gfCNCPoint6[3646] = {X 38.0615, Y 40.7422, Z -8.0000, A 0.000, B 0.000, C 0.000 }
gfCNCPoint6[3647] = {X 38.9310, Y 40.2409, Z -8.0000, A 0.000, B 0.000, C 0.000 }
gfCNCPoint6[3648] = {X 39.5220, Y 38.8450, Z -8.0000, A 0.000, B 0.000, C 0.000 }
gfCNCPoint6[3649] = {X 40.0631, Y 37.4290, Z -8.0000, A 0.000, B 0.000, C 0.000 }
gfCNCPoint6[3650] = {X 43.6474, Y 27.8074, Z -8.0000, A 0.000, B 0.000, C 0.000 }
gfCNCPoint6[3651] = {X 39.8991, Y 26.4111, Z -8.0000, A 0.000, B 0.000, C 0.000 }
gfCNCPoint6[3652] = {X 43.7224, Y 27.8353, Z -8.0000, A 0.000, B 0.000, C 0.000 }
gfCNCPoint6[3653] = {X 48.3793, Y 15.3344, Z -8.0000, A 0.000, B 0.000, C 0.000 }
gfCNCPoint6[3654] = {X 47.9922, Y 14.6130, Z -8.0000, A 0.000, B 0.000, C 0.000 }
gfCNCPoint6[3655] = {X 47.7508, Y 13.8307, Z -8.0000, A 0.000, B 0.000, C 0.000 }
gfCNCPoint6[3656] = {X 47.6644, Y 13.0166, Z -8.0000, A 0.000, B 0.000, C 0.000 }
gfCNCPoint6[3657] = {X 47.6642, Y 12.1868, Z -8.0000, A 0.000, B 0.000, C 0.000 }
gfCNCPoint6[3658] = {X 47.7705, Y 11.2433, Z -8.0000, A 0.000, B 0.000, C 0.000 }
gfCNCPoint6[3659] = {X 48.0841, Y 10.3472, Z -8.0000, A 0.000, B 0.000, C 0.000 }
gfCNCPoint6[3660] = {X 48.5893, Y 9.5432, Z -8.0000, A 0.000, B 0.000, C 0.000 }
gfCNCPoint6[3661] = {X 49.2606, Y 8.8719, Z -8.0000, A 0.000, B 0.000, C 0.000 }
gfCNCPoint6[3662] = {X 50.0646, Y 8.3667, Z -8.0000, A 0.000, B 0.000, C 0.000 }
gfCNCPoint6[3663] = {X 50.9607, Y 8.0531, Z -8.0000, A 0.000, B 0.000, C 0.000 }
gfCNCPoint6[3664] = {X 51.9042, Y 7.9468, Z -8.0000, A 0.000, B 0.000, C 0.000 }
gfCNCPoint6[3665] = {X 59.6221, Y 7.9468, Z -8.0000, A 0.000, B 0.000, C 0.000 }
gfCNCPoint6[3666] = {X 60.5656, Y 8.0531, Z -8.0000, A 0.000, B 0.000, C 0.000 }
gfCNCPoint6[3667] = {X 61.4618, Y 8.3667, Z -8.0000, A 0.000, B 0.000, C 0.000 }
gfCNCPoint6[3668] = {X 62.2657, Y 8.8718, Z -8.0000, A 0.000, B 0.000, C 0.000 }
gfCNCPoint6[3669] = {X 62.9371, Y 9.5432, Z -8.0000, A 0.000, B 0.000, C 0.000 }
gfCNCPoint6[3670] = {X 63.4422, Y 10.3471, Z -8.0000, A 0.000, B 0.000, C 0.000 }
gfCNCPoint6[3671] = {X 63.7558, Y 11.2433, Z -8.0000, A 0.000, B 0.000, C 0.000 }
gfCNCPoint6[3672] = {X 63.8621, Y 12.1868, Z -8.0000, A 0.000, B 0.000, C 0.000 }
gfCNCPoint6[3673] = {X 63.8621, Y 12.9782, Z -8.0000, A 0.000, B 0.000, C 0.000 }
gfCNCPoint6[3674] = {X 63.7772, Y 13.8222, Z -8.0000, A 0.000, B 0.000, C 0.000 }
gfCNCPoint6[3675] = {X 63.5261, Y 14.6323, Z -8.0000, A 0.000, B 0.000, C 0.000 }
gfCNCPoint6[3676] = {X 63.1187, Y 15.3763, Z -8.0000, A 0.000, B 0.000, C 0.000 }
gfCNCPoint6[3677] = {X 63.3523, Y 15.9915, Z -8.0000, A 0.000, B 0.000, C 0.000 }
gfCNCPoint6[3678] = {X 66.1652, Y 23.4578, Z -8.0000, A 0.000, B 0.000, C 0.000 }
gfCNCPoint6[3679] = {X 72.1363, Y 39.5291, Z -8.0000, A 0.000, B 0.000, C 0.000 }
gfCNCPoint6[3680] = {X 72.4543, Y 40.3288, Z -8.0000, A 0.000, B 0.000, C 0.000 }
gfCNCPoint6[3681] = {X 73.2915, Y 40.8190, Z -8.0000, A 0.000, B 0.000, C 0.000 }
gfCNCPoint6[3682] = {X 73.9953, Y 41.4867, Z -8.0000, A 0.000, B 0.000, C 0.000 }
gfCNCPoint6[3683] = {X 74.5289, Y 42.2969, Z -8.0000, A 0.000, B 0.000, C 0.000 }
gfCNCPoint6[3684] = {X 74.8645, Y 43.2072, Z -8.0000, A 0.000, B 0.000, C 0.000 }
gfCNCPoint6[3685] = {X 74.9843, Y 44.1699, Z -8.0000, A 0.000, B 0.000, C 0.000 }
gfCNCPoint6[3686] = {X 74.9845, Y 45.0000, Z -8.0000, A 0.000, B 0.000, C 0.000 }
gfCNCPoint6[3687] = {X 74.8782, Y 45.9435, Z -8.0000, A 0.000, B 0.000, C 0.000 }
gfCNCPoint6[3688] = {X 74.5646, Y 46.8397, Z -8.0000, A 0.000, B 0.000, C 0.000 }
gfCNCPoint6[3689] = {X 74.0594, Y 47.6436, Z -8.0000, A 0.000, B 0.000, C 0.000 }
gfCNCPoint6[3690] = {X 73.3881, Y 48.3150, Z -8.0000, A 0.000, B 0.000, C 0.000 }
gfCNCPoint6[3691] = {X 72.5841, Y 48.8201, Z -8.0000, A 0.000, B 0.000, C 0.000 }
gfCNCPoint6[3692] = {X 71.6879, Y 49.1337, Z -8.0000, A 0.000, B 0.000, C 0.000 }
gfCNCPoint6[3693] = {X 70.7445, Y 49.2400, Z -8.0000, A 0.000, B 0.000, C 0.000 }
gfCNCPoint6[3694] = {X 64.1851, Y 49.2400, Z -8.0000, A 0.000, B 0.000, C 0.000 }
gfCNCPoint6[3695] = {X 63.2416, Y 49.1337, Z -8.0000, A 0.000, B 0.000, C 0.000 }
gfCNCPoint6[3696] = {X 62.3455, Y 48.8201, Z -8.0000, A 0.000, B 0.000, C 0.000 }
gfCNCPoint6[3697] = {X 61.5415, Y 48.3150, Z -8.0000, A 0.000, B 0.000, C 0.000 }
gfCNCPoint6[3698] = {X 60.8702, Y 47.6436, Z -8.0000, A 0.000, B 0.000, C 0.000 }
gfCNCPoint6[3699] = {X 60.3650, Y 46.8397, Z -8.0000, A 0.000, B 0.000, C 0.000 }
gfCNCPoint6[3700] = {X 60.0514, Y 45.9435, Z -8.0000, A 0.000, B 0.000, C 0.000 }
gfCNCPoint6[3701] = {X 59.9451, Y 45.0000, Z -8.0000, A 0.000, B 0.000, C 0.000 }
gfCNCPoint6[3702] = {X 59.9451, Y 44.2085, Z -8.0000, A 0.000, B 0.000, C 0.000 }
gfCNCPoint6[3703] = {X 60.0327, Y 43.3528, Z -8.0000, A 0.000, B 0.000, C 0.000 }
gfCNCPoint6[3704] = {X 60.2911, Y 42.5324, Z -8.0000, A 0.000, B 0.000, C 0.000 }
gfCNCPoint6[3705] = {X 60.7098, Y 41.7810, Z -8.0000, A 0.000, B 0.000, C 0.000 }
gfCNCPoint6[3706] = {X 60.0623, Y 40.0092, Z -8.0000, A 0.000, B 0.000, C 0.000 }
gfCNCPoint6[3707] = {X 52.0229, Y 40.0092, Z -8.0000, A 0.000, B 0.000, C 0.000 }
gfCNCPoint6[3708] = {X 51.2471, Y 42.0939, Z -8.0000, A 0.000, B 0.000, C 0.000 }
gfCNCPoint6[3709] = {X 51.2689, Y 42.1309, Z -8.0000, A 0.000, B 0.000, C 0.000 }
gfCNCPoint6[3710] = {X 51.5641, Y 42.7777, Z -8.0000, A 0.000, B 0.000, C 0.000 }
gfCNCPoint6[3711] = {X 51.7471, Y 43.4647, Z -8.0000, A 0.000, B 0.000, C 0.000 }
gfCNCPoint6[3712] = {X 51.8128, Y 44.1726, Z -8.0000, A 0.000, B 0.000, C 0.000 }
gfCNCPoint6[3713] = {X 51.8129, Y 45.0000, Z -8.0000, A 0.000, B 0.000, C 0.000 }
gfCNCPoint6[3714] = {X 51.7066, Y 45.9435, Z -8.0000, A 0.000, B 0.000, C 0.000 }
gfCNCPoint6[3715] = {X 51.3930, Y 46.8397, Z -8.0000, A 0.000, B 0.000, C 0.000 }
gfCNCPoint6[3716] = {X 50.8879, Y 47.6436, Z -8.0000, A 0.000, B 0.000, C 0.000 }
gfCNCPoint6[3717] = {X 50.2165, Y 48.3150, Z -8.0000, A 0.000, B 0.000, C 0.000 }
gfCNCPoint6[3718] = {X 49.4126, Y 48.8201, Z -8.0000, A 0.000, B 0.000, C 0.000 }
gfCNCPoint6[3719] = {X 48.5164, Y 49.1337, Z -8.0000, A 0.000, B 0.000, C 0.000 }
gfCNCPoint6[3720] = {X 47.5729, Y 49.2400, Z -8.0000, A 0.000, B 0.000, C 0.000 }
gfCNCPoint6[3721] = {X 40.6393, Y 49.2400, Z -8.0000, A 0.000, B 0.000, C 0.000 }
gfCNCPoint6[3722] = {X 39.6958, Y 49.1337, Z -8.0000, A 0.000, B 0.000, C 0.000 }
gfCNCPoint6[3723] = {X 38.7996, Y 48.8201, Z -8.0000, A 0.000, B 0.000, C 0.000 }
gfCNCPoint6[3724] = {X 37.9957, Y 48.3150, Z -8.0000, A 0.000, B 0.000, C 0.000 }
gfCNCPoint6[3725] = {X 37.3243, Y 47.6436, Z -8.0000, A 0.000, B 0.000, C 0.000 }
gfCNCPoint6[3726] = {X 36.8192, Y 46.8397, Z -8.0000, A 0.000, B 0.000, C 0.000 }
gfCNCPoint6[3727] = {X 36.5056, Y 45.9435, Z -8.0000, A 0.000, B 0.000, C 0.000 }
gfCNCPoint6[3728] = {X 36.3993, Y 45.0000, Z -8.0000, A 0.000, B 0.000, C 0.000 }
gfCNCPoint6[3729] = {X 36.3993, Y 44.2086, Z -8.0000, A 0.000, B 0.000, C 0.000 }
gfCNCPoint6[3730] = {X 36.5152, Y 43.2242, Z -8.0000, A 0.000, B 0.000, C 0.000 }
gfCNCPoint6[3731] = {X 36.8565, Y 42.2936, Z -8.0000, A 0.000, B 0.000, C 0.000 }
gfCNCPoint6[3732] = {X 37.4045, Y 41.4677, Z -8.0000, A 0.000, B 0.000, C 0.000 }
gfCNCPoint6[3733] = {X 38.1293, Y 40.7916, Z -8.0000, A 0.000, B 0.000, C 0.000 }
gfCNCPoint6[3734] = {X 38.9913, Y 40.3022, Z -8.0000, A 0.000, B 0.000, C 0.000 }
gfCNCPoint6[3735] = {X 39.5904, Y 38.8895, Z -8.0000, A 0.000, B 0.000, C 0.000 }
gfCNCPoint6[3736] = {X 40.1384, Y 37.4563, Z -8.0000, A 0.000, B 0.000, C 0.000 }
gfCNCPoint6[3737] = {X 43.7224, Y 27.8353, Z -8.0000, A 0.000, B 0.000, C 0.000 }
gfCNCPoint6[3738] = {X 39.9740, Y 26.4390, Z -8.0000, A 0.000, B 0.000, C 0.000 }
gfCNCPoint6[3739] = {X 43.7974, Y 27.8633, Z -8.0000, A 0.000, B 0.000, C 0.000 }
gfCNCPoint6[3740] = {X 48.4687, Y 15.3238, Z -8.0000, A 0.000, B 0.000, C 0.000 }
gfCNCPoint6[3741] = {X 48.0765, Y 14.6072, Z -8.0000, A 0.000, B 0.000, C 0.000 }
gfCNCPoint6[3742] = {X 47.8320, Y 13.8279, Z -8.0000, A 0.000, B 0.000, C 0.000 }
gfCNCPoint6[3743] = {X 47.7444, Y 13.0158, Z -8.0000, A 0.000, B 0.000, C 0.000 }
gfCNCPoint6[3744] = {X 47.7442, Y 12.1868, Z -8.0000, A 0.000, B 0.000, C 0.000 }
gfCNCPoint6[3745] = {X 47.8485, Y 11.2611, Z -8.0000, A 0.000, B 0.000, C 0.000 }
gfCNCPoint6[3746] = {X 48.1562, Y 10.3819, Z -8.0000, A 0.000, B 0.000, C 0.000 }
gfCNCPoint6[3747] = {X 48.6518, Y 9.5931, Z -8.0000, A 0.000, B 0.000, C 0.000 }
gfCNCPoint6[3748] = {X 49.3105, Y 8.9344, Z -8.0000, A 0.000, B 0.000, C 0.000 }
gfCNCPoint6[3749] = {X 50.0993, Y 8.4388, Z -8.0000, A 0.000, B 0.000, C 0.000 }
gfCNCPoint6[3750] = {X 50.9785, Y 8.1311, Z -8.0000, A 0.000, B 0.000, C 0.000 }
gfCNCPoint6[3751] = {X 51.9042, Y 8.0268, Z -8.0000, A 0.000, B 0.000, C 0.000 }
gfCNCPoint6[3752] = {X 59.6221, Y 8.0268, Z -8.0000, A 0.000, B 0.000, C 0.000 }
gfCNCPoint6[3753] = {X 60.5478, Y 8.1311, Z -8.0000, A 0.000, B 0.000, C 0.000 }
gfCNCPoint6[3754] = {X 61.4271, Y 8.4388, Z -8.0000, A 0.000, B 0.000, C 0.000 }
gfCNCPoint6[3755] = {X 62.2158, Y 8.9344, Z -8.0000, A 0.000, B 0.000, C 0.000 }
gfCNCPoint6[3756] = {X 62.8745, Y 9.5931, Z -8.0000, A 0.000, B 0.000, C 0.000 }
gfCNCPoint6[3757] = {X 63.3702, Y 10.3819, Z -8.0000, A 0.000, B 0.000, C 0.000 }
gfCNCPoint6[3758] = {X 63.6778, Y 11.2611, Z -8.0000, A 0.000, B 0.000, C 0.000 }
gfCNCPoint6[3759] = {X 63.7821, Y 12.1868, Z -8.0000, A 0.000, B 0.000, C 0.000 }
gfCNCPoint6[3760] = {X 63.7821, Y 12.9782, Z -8.0000, A 0.000, B 0.000, C 0.000 }
gfCNCPoint6[3761] = {X 63.6961, Y 13.8198, Z -8.0000, A 0.000, B 0.000, C 0.000 }
gfCNCPoint6[3762] = {X 63.4415, Y 14.6267, Z -8.0000, A 0.000, B 0.000, C 0.000 }
gfCNCPoint6[3763] = {X 63.0289, Y 15.3654, Z -8.0000, A 0.000, B 0.000, C 0.000 }
gfCNCPoint6[3764] = {X 63.2774, Y 16.0198, Z -8.0000, A 0.000, B 0.000, C 0.000 }
gfCNCPoint6[3765] = {X 66.0903, Y 23.4859, Z -8.0000, A 0.000, B 0.000, C 0.000 }
gfCNCPoint6[3766] = {X 72.0617, Y 39.5578, Z -8.0000, A 0.000, B 0.000, C 0.000 }
gfCNCPoint6[3767] = {X 72.3921, Y 40.3890, Z -8.0000, A 0.000, B 0.000, C 0.000 }
gfCNCPoint6[3768] = {X 73.2225, Y 40.8674, Z -8.0000, A 0.000, B 0.000, C 0.000 }
gfCNCPoint6[3769] = {X 73.9214, Y 41.5231, Z -8.0000, A 0.000, B 0.000, C 0.000 }
gfCNCPoint6[3770] = {X 74.4516, Y 42.3213, Z -8.0000, A 0.000, B 0.000, C 0.000 }
gfCNCPoint6[3771] = {X 74.7852, Y 43.2197, Z -8.0000, A 0.000, B 0.000, C 0.000 }
gfCNCPoint6[3772] = {X 74.9043, Y 44.1706, Z -8.0000, A 0.000, B 0.000, C 0.000 }
gfCNCPoint6[3773] = {X 74.9045, Y 45.0000, Z -8.0000, A 0.000, B 0.000, C 0.000 }
gfCNCPoint6[3774] = {X 74.8002, Y 45.9257, Z -8.0000, A 0.000, B 0.000, C 0.000 }
gfCNCPoint6[3775] = {X 74.4925, Y 46.8050, Z -8.0000, A 0.000, B 0.000, C 0.000 }
gfCNCPoint6[3776] = {X 73.9969, Y 47.5937, Z -8.0000, A 0.000, B 0.000, C 0.000 }
gfCNCPoint6[3777] = {X 73.3382, Y 48.2524, Z -8.0000, A 0.000, B 0.000, C 0.000 }
gfCNCPoint6[3778] = {X 72.5494, Y 48.7480, Z -8.0000, A 0.000, B 0.000, C 0.000 }
gfCNCPoint6[3779] = {X 71.6701, Y 49.0557, Z -8.0000, A 0.000, B 0.000, C 0.000 }
gfCNCPoint6[3780] = {X 70.7445, Y 49.1600, Z -8.0000, A 0.000, B 0.000, C 0.000 }
gfCNCPoint6[3781] = {X 64.1851, Y 49.1600, Z -8.0000, A 0.000, B 0.000, C 0.000 }
gfCNCPoint6[3782] = {X 63.2594, Y 49.0557, Z -8.0000, A 0.000, B 0.000, C 0.000 }
gfCNCPoint6[3783] = {X 62.3802, Y 48.7480, Z -8.0000, A 0.000, B 0.000, C 0.000 }
gfCNCPoint6[3784] = {X 61.5914, Y 48.2524, Z -8.0000, A 0.000, B 0.000, C 0.000 }
gfCNCPoint6[3785] = {X 60.9327, Y 47.5937, Z -8.0000, A 0.000, B 0.000, C 0.000 }
gfCNCPoint6[3786] = {X 60.4371, Y 46.8050, Z -8.0000, A 0.000, B 0.000, C 0.000 }
gfCNCPoint6[3787] = {X 60.1294, Y 45.9257, Z -8.0000, A 0.000, B 0.000, C 0.000 }
gfCNCPoint6[3788] = {X 60.0251, Y 45.0000, Z -8.0000, A 0.000, B 0.000, C 0.000 }
gfCNCPoint6[3789] = {X 60.0251, Y 44.2086, Z -8.0000, A 0.000, B 0.000, C 0.000 }
gfCNCPoint6[3790] = {X 60.1139, Y 43.3555, Z -8.0000, A 0.000, B 0.000, C 0.000 }
gfCNCPoint6[3791] = {X 60.3756, Y 42.5387, Z -8.0000, A 0.000, B 0.000, C 0.000 }
gfCNCPoint6[3792] = {X 60.7994, Y 41.7930, Z -8.0000, A 0.000, B 0.000, C 0.000 }
gfCNCPoint6[3793] = {X 60.1182, Y 39.9292, Z -8.0000, A 0.000, B 0.000, C 0.000 }
gfCNCPoint6[3794] = {X 51.9673, Y 39.9292, Z -8.0000, A 0.000, B 0.000, C 0.000 }
gfCNCPoint6[3795] = {X 51.1588, Y 42.1017, Z -8.0000, A 0.000, B 0.000, C 0.000 }
gfCNCPoint6[3796] = {X 51.1995, Y 42.1708, Z -8.0000, A 0.000, B 0.000, C 0.000 }
gfCNCPoint6[3797] = {X 51.4890, Y 42.8052, Z -8.0000, A 0.000, B 0.000, C 0.000 }
gfCNCPoint6[3798] = {X 51.6684, Y 43.4790, Z -8.0000, A 0.000, B 0.000, C 0.000 }
gfCNCPoint6[3799] = {X 51.7328, Y 44.1733, Z -8.0000, A 0.000, B 0.000, C 0.000 }
gfCNCPoint6[3800] = {X 51.7329, Y 45.0000, Z -8.0000, A 0.000, B 0.000, C 0.000 }
gfCNCPoint6[3801] = {X 51.6286, Y 45.9257, Z -8.0000, A 0.000, B 0.000, C 0.000 }
gfCNCPoint6[3802] = {X 51.3210, Y 46.8050, Z -8.0000, A 0.000, B 0.000, C 0.000 }
gfCNCPoint6[3803] = {X 50.8253, Y 47.5937, Z -8.0000, A 0.000, B 0.000, C 0.000 }
gfCNCPoint6[3804] = {X 50.1666, Y 48.2524, Z -8.0000, A 0.000, B 0.000, C 0.000 }
gfCNCPoint6[3805] = {X 49.3779, Y 48.7480, Z -8.0000, A 0.000, B 0.000, C 0.000 }
gfCNCPoint6[3806] = {X 48.4986, Y 49.0557, Z -8.0000, A 0.000, B 0.000, C 0.000 }
gfCNCPoint6[3807] = {X 47.5729, Y 49.1600, Z -8.0000, A 0.000, B 0.000, C 0.000 }
gfCNCPoint6[3808] = {X 40.6393, Y 49.1600, Z -8.0000, A 0.000, B 0.000, C 0.000 }
gfCNCPoint6[3809] = {X 39.7136, Y 49.0557, Z -8.0000, A 0.000, B 0.000, C 0.000 }
gfCNCPoint6[3810] = {X 38.8343, Y 48.7480, Z -8.0000, A 0.000, B 0.000, C 0.000 }
gfCNCPoint6[3811] = {X 38.0456, Y 48.2524, Z -8.0000, A 0.000, B 0.000, C 0.000 }
gfCNCPoint6[3812] = {X 37.3869, Y 47.5937, Z -8.0000, A 0.000, B 0.000, C 0.000 }
gfCNCPoint6[3813] = {X 36.8913, Y 46.8050, Z -8.0000, A 0.000, B 0.000, C 0.000 }
gfCNCPoint6[3814] = {X 36.5836, Y 45.9257, Z -8.0000, A 0.000, B 0.000, C 0.000 }
gfCNCPoint6[3815] = {X 36.4793, Y 45.0000, Z -8.0000, A 0.000, B 0.000, C 0.000 }
gfCNCPoint6[3816] = {X 36.4793, Y 44.2086, Z -8.0000, A 0.000, B 0.000, C 0.000 }
gfCNCPoint6[3817] = {X 36.5945, Y 43.2366, Z -8.0000, A 0.000, B 0.000, C 0.000 }
gfCNCPoint6[3818] = {X 36.9336, Y 42.3185, Z -8.0000, A 0.000, B 0.000, C 0.000 }
gfCNCPoint6[3819] = {X 37.4778, Y 41.5050, Z -8.0000, A 0.000, B 0.000, C 0.000 }
gfCNCPoint6[3820] = {X 38.1970, Y 40.8412, Z -8.0000, A 0.000, B 0.000, C 0.000 }
gfCNCPoint6[3821] = {X 39.0514, Y 40.3638, Z -8.0000, A 0.000, B 0.000, C 0.000 }
gfCNCPoint6[3822] = {X 39.6586, Y 38.9342, Z -8.0000, A 0.000, B 0.000, C 0.000 }
gfCNCPoint6[3823] = {X 40.2136, Y 37.4835, Z -8.0000, A 0.000, B 0.000, C 0.000 }
gfCNCPoint6[3824] = {X 43.7974, Y 27.8633, Z -8.0000, A 0.000, B 0.000, C 0.000 }
gfCNCPoint6[3825] = {X 40.0490, Y 26.4669, Z -8.0000, A 0.000, B 0.000, C 0.000 }
gfCNCPoint6[3826] = {X 43.8723, Y 27.8912, Z -8.0000, A 0.000, B 0.000, C 0.000 }
gfCNCPoint6[3827] = {X 48.5582, Y 15.3126, Z -8.0000, A 0.000, B 0.000, C 0.000 }
gfCNCPoint6[3828] = {X 48.1610, Y 14.6012, Z -8.0000, A 0.000, B 0.000, C 0.000 }
gfCNCPoint6[3829] = {X 47.9131, Y 13.8250, Z -8.0000, A 0.000, B 0.000, C 0.000 }
gfCNCPoint6[3830] = {X 47.8244, Y 13.0151, Z -8.0000, A 0.000, B 0.000, C 0.000 }
gfCNCPoint6[3831] = {X 47.8242, Y 12.1868, Z -8.0000, A 0.000, B 0.000, C 0.000 }
gfCNCPoint6[3832] = {X 47.9265, Y 11.2789, Z -8.0000, A 0.000, B 0.000, C 0.000 }
gfCNCPoint6[3833] = {X 48.2283, Y 10.4166, Z -8.0000, A 0.000, B 0.000, C 0.000 }
gfCNCPoint6[3834] = {X 48.7144, Y 9.6430, Z -8.0000, A 0.000, B 0.000, C 0.000 }
gfCNCPoint6[3835] = {X 49.3604, Y 8.9969, Z -8.0000, A 0.000, B 0.000, C 0.000 }
gfCNCPoint6[3836] = {X 50.1340, Y 8.5109, Z -8.0000, A 0.000, B 0.000, C 0.000 }
gfCNCPoint6[3837] = {X 50.9963, Y 8.2091, Z -8.0000, A 0.000, B 0.000, C 0.000 }
gfCNCPoint6[3838] = {X 51.9042, Y 8.1068, Z -8.0000, A 0.000, B 0.000, C 0.000 }
gfCNCPoint6[3839] = {X 59.6221, Y 8.1068, Z -8.0000, A 0.000, B 0.000, C 0.000 }
gfCNCPoint6[3840] = {X 60.5300, Y 8.2091, Z -8.0000, A 0.000, B 0.000, C 0.000 }
gfCNCPoint6[3841] = {X 61.3924, Y 8.5109, Z -8.0000, A 0.000, B 0.000, C 0.000 }
gfCNCPoint6[3842] = {X 62.1660, Y 8.9969, Z -8.0000, A 0.000, B 0.000, C 0.000 }
gfCNCPoint6[3843] = {X 62.8120, Y 9.6430, Z -8.0000, A 0.000, B 0.000, C 0.000 }
gfCNCPoint6[3844] = {X 63.2981, Y 10.4166, Z -8.0000, A 0.000, B 0.000, C 0.000 }
gfCNCPoint6[3845] = {X 63.5998, Y 11.2789, Z -8.0000, A 0.000, B 0.000, C 0.000 }
gfCNCPoint6[3846] = {X 63.7021, Y 12.1868, Z -8.0000, A 0.000, B 0.000, C 0.000 }
gfCNCPoint6[3847] = {X 63.7021, Y 12.9782, Z -8.0000, A 0.000, B 0.000, C 0.000 }
gfCNCPoint6[3848] = {X 63.6148, Y 13.8174, Z -8.0000, A 0.000, B 0.000, C 0.000 }
gfCNCPoint6[3849] = {X 63.3568, Y 14.6208, Z -8.0000, A 0.000, B 0.000, C 0.000 }
gfCNCPoint6[3850] = {X 62.9390, Y 15.3539, Z -8.0000, A 0.000, B 0.000, C 0.000 }
gfCNCPoint6[3851] = {X 63.2026, Y 16.0481, Z -8.0000, A 0.000, B 0.000, C 0.000 }
gfCNCPoint6[3852] = {X 66.0153, Y 23.5139, Z -8.0000, A 0.000, B 0.000, C 0.000 }
gfCNCPoint6[3853] = {X 71.9870, Y 39.5865, Z -8.0000, A 0.000, B 0.000, C 0.000 }
gfCNCPoint6[3854] = {X 72.3301, Y 40.4495, Z -8.0000, A 0.000, B 0.000, C 0.000 }
gfCNCPoint6[3855] = {X 73.1536, Y 40.9160, Z -8.0000, A 0.000, B 0.000, C 0.000 }
gfCNCPoint6[3856] = {X 73.8474, Y 41.5597, Z -8.0000, A 0.000, B 0.000, C 0.000 }
gfCNCPoint6[3857] = {X 74.3743, Y 42.3459, Z -8.0000, A 0.000, B 0.000, C 0.000 }
gfCNCPoint6[3858] = {X 74.7059, Y 43.2324, Z -8.0000, A 0.000, B 0.000, C 0.000 }
gfCNCPoint6[3859] = {X 74.8243, Y 44.1714, Z -8.0000, A 0.000, B 0.000, C 0.000 }
gfCNCPoint6[3860] = {X 74.8245, Y 45.0000, Z -8.0000, A 0.000, B 0.000, C 0.000 }
gfCNCPoint6[3861] = {X 74.7222, Y 45.9079, Z -8.0000, A 0.000, B 0.000, C 0.000 }
gfCNCPoint6[3862] = {X 74.4204, Y 46.7702, Z -8.0000, A 0.000, B 0.000, C 0.000 }
gfCNCPoint6[3863] = {X 73.9343, Y 47.5438, Z -8.0000, A 0.000, B 0.000, C 0.000 }
gfCNCPoint6[3864] = {X 73.2883, Y 48.1899, Z -8.0000, A 0.000, B 0.000, C 0.000 }
gfCNCPoint6[3865] = {X 72.5147, Y 48.6760, Z -8.0000, A 0.000, B 0.000, C 0.000 }
gfCNCPoint6[3866] = {X 71.6523, Y 48.9777, Z -8.0000, A 0.000, B 0.000, C 0.000 }
gfCNCPoint6[3867] = {X 70.7445, Y 49.0800, Z -8.0000, A 0.000, B 0.000, C 0.000 }
gfCNCPoint6[3868] = {X 64.1851, Y 49.0800, Z -8.0000, A 0.000, B 0.000, C 0.000 }
gfCNCPoint6[3869] = {X 63.2772, Y 48.9777, Z -8.0000, A 0.000, B 0.000, C 0.000 }
gfCNCPoint6[3870] = {X 62.4149, Y 48.6760, Z -8.0000, A 0.000, B 0.000, C 0.000 }
gfCNCPoint6[3871] = {X 61.6413, Y 48.1899, Z -8.0000, A 0.000, B 0.000, C 0.000 }
gfCNCPoint6[3872] = {X 60.9953, Y 47.5438, Z -8.0000, A 0.000, B 0.000, C 0.000 }
gfCNCPoint6[3873] = {X 60.5092, Y 46.7702, Z -8.0000, A 0.000, B 0.000, C 0.000 }
gfCNCPoint6[3874] = {X 60.2074, Y 45.9079, Z -8.0000, A 0.000, B 0.000, C 0.000 }
gfCNCPoint6[3875] = {X 60.1051, Y 45.0000, Z -8.0000, A 0.000, B 0.000, C 0.000 }
gfCNCPoint6[3876] = {X 60.1051, Y 44.2086, Z -8.0000, A 0.000, B 0.000, C 0.000 }
gfCNCPoint6[3877] = {X 60.1950, Y 43.3582, Z -8.0000, A 0.000, B 0.000, C 0.000 }
gfCNCPoint6[3878] = {X 60.4602, Y 42.5452, Z -8.0000, A 0.000, B 0.000, C 0.000 }
gfCNCPoint6[3879] = {X 60.8891, Y 41.8054, Z -8.0000, A 0.000, B 0.000, C 0.000 }
gfCNCPoint6[3880] = {X 60.1742, Y 39.8492, Z -8.0000, A 0.000, B 0.000, C 0.000 }
gfCNCPoint6[3881] = {X 51.9117, Y 39.8492, Z -8.0000, A 0.000, B 0.000, C 0.000 }
gfCNCPoint6[3882] = {X 51.0705, Y 42.1095, Z -8.0000, A 0.000, B 0.000, C 0.000 }
gfCNCPoint6[3883] = {X 51.1302, Y 42.2107, Z -8.0000, A 0.000, B 0.000, C 0.000 }
gfCNCPoint6[3884] = {X 51.4139, Y 42.8327, Z -8.0000, A 0.000, B 0.000, C 0.000 }
gfCNCPoint6[3885] = {X 51.5897, Y 43.4933, Z -8.0000, A 0.000, B 0.000, C 0.000 }
gfCNCPoint6[3886] = {X 51.6528, Y 44.1740, Z -8.0000, A 0.000, B 0.000, C 0.000 }
gfCNCPoint6[3887] = {X 51.6529, Y 45.0000, Z -8.0000, A 0.000, B 0.000, C 0.000 }
gfCNCPoint6[3888] = {X 51.5506, Y 45.9079, Z -8.0000, A 0.000, B 0.000, C 0.000 }
gfCNCPoint6[3889] = {X 51.2489, Y 46.7702, Z -8.0000, A 0.000, B 0.000, C 0.000 }
gfCNCPoint6[3890] = {X 50.7628, Y 47.5438, Z -8.0000, A 0.000, B 0.000, C 0.000 }
gfCNCPoint6[3891] = {X 50.1168, Y 48.1899, Z -8.0000, A 0.000, B 0.000, C 0.000 }
gfCNCPoint6[3892] = {X 49.3432, Y 48.6760, Z -8.0000, A 0.000, B 0.000, C 0.000 }
gfCNCPoint6[3893] = {X 48.4808, Y 48.9777, Z -8.0000, A 0.000, B 0.000, C 0.000 }
gfCNCPoint6[3894] = {X 47.5729, Y 49.0800, Z -8.0000, A 0.000, B 0.000, C 0.000 }
gfCNCPoint6[3895] = {X 40.6393, Y 49.0800, Z -8.0000, A 0.000, B 0.000, C 0.000 }
gfCNCPoint6[3896] = {X 39.7314, Y 48.9777, Z -8.0000, A 0.000, B 0.000, C 0.000 }
gfCNCPoint6[3897] = {X 38.8691, Y 48.6760, Z -8.0000, A 0.000, B 0.000, C 0.000 }
gfCNCPoint6[3898] = {X 38.0955, Y 48.1899, Z -8.0000, A 0.000, B 0.000, C 0.000 }
gfCNCPoint6[3899] = {X 37.4494, Y 47.5438, Z -8.0000, A 0.000, B 0.000, C 0.000 }
gfCNCPoint6[3900] = {X 36.9633, Y 46.7702, Z -8.0000, A 0.000, B 0.000, C 0.000 }
gfCNCPoint6[3901] = {X 36.6616, Y 45.9079, Z -8.0000, A 0.000, B 0.000, C 0.000 }
gfCNCPoint6[3902] = {X 36.5593, Y 45.0000, Z -8.0000, A 0.000, B 0.000, C 0.000 }
gfCNCPoint6[3903] = {X 36.5593, Y 44.2086, Z -8.0000, A 0.000, B 0.000, C 0.000 }
gfCNCPoint6[3904] = {X 36.6733, Y 43.2512, Z -8.0000, A 0.000, B 0.000, C 0.000 }
gfCNCPoint6[3905] = {X 37.0087, Y 42.3474, Z -8.0000, A 0.000, B 0.000, C 0.000 }
gfCNCPoint6[3906] = {X 37.5468, Y 41.5474, Z -8.0000, A 0.000, B 0.000, C 0.000 }
gfCNCPoint6[3907] = {X 38.2576, Y 40.8961, Z -8.0000, A 0.000, B 0.000, C 0.000 }
gfCNCPoint6[3908] = {X 39.1014, Y 40.4297, Z -8.0000, A 0.000, B 0.000, C 0.000 }
gfCNCPoint6[3909] = {X 39.1158, Y 40.4158, Z -8.0000, A 0.000, B 0.000, C 0.000 }
gfCNCPoint6[3910] = {X 39.1244, Y 40.3964, Z -8.0000, A 0.000, B 0.000, C 0.000 }
gfCNCPoint6[3911] = {X 39.7328, Y 38.9641, Z -8.0000, A 0.000, B 0.000, C 0.000 }
gfCNCPoint6[3912] = {X 40.2888, Y 37.5107, Z -8.0000, A 0.000, B 0.000, C 0.000 }
gfCNCPoint6[3913] = {X 43.8723, Y 27.8912, Z -8.0000, A 0.000, B 0.000, C 0.000 }
gfCNCPoint6[3914] = {X 40.1240, Y 26.4948, Z -8.0000, A 0.000, B 0.000, C 0.000 }
gfCNCPoint6[3915] = {X 43.9473, Y 27.9191, Z -8.0000, A 0.000, B 0.000, C 0.000 }
gfCNCPoint6[3916] = {X 48.6479, Y 15.3010, Z -8.0000, A 0.000, B 0.000, C 0.000 }
gfCNCPoint6[3917] = {X 48.2407, Y 14.5838, Z -8.0000, A 0.000, B 0.000, C 0.000 }
gfCNCPoint6[3918] = {X 47.9892, Y 13.7983, Z -8.0000, A 0.000, B 0.000, C 0.000 }
gfCNCPoint6[3919] = {X 47.9042, Y 12.9780, Z -8.0000, A 0.000, B 0.000, C 0.000 }
gfCNCPoint6[3920] = {X 47.9042, Y 12.1868, Z -8.0000, A 0.000, B 0.000, C 0.000 }
gfCNCPoint6[3921] = {X 48.0045, Y 11.2967, Z -8.0000, A 0.000, B 0.000, C 0.000 }
gfCNCPoint6[3922] = {X 48.3003, Y 10.4513, Z -8.0000, A 0.000, B 0.000, C 0.000 }
gfCNCPoint6[3923] = {X 48.7769, Y 9.6929, Z -8.0000, A 0.000, B 0.000, C 0.000 }
gfCNCPoint6[3924] = {X 49.4103, Y 9.0595, Z -8.0000, A 0.000, B 0.000, C 0.000 }
gfCNCPoint6[3925] = {X 50.1687, Y 8.5829, Z -8.0000, A 0.000, B 0.000, C 0.000 }
gfCNCPoint6[3926] = {X 51.0141, Y 8.2871, Z -8.0000, A 0.000, B 0.000, C 0.000 }
gfCNCPoint6[3927] = {X 51.9042, Y 8.1868, Z -8.0000, A 0.000, B 0.000, C 0.000 }
gfCNCPoint6[3928] = {X 59.6221, Y 8.1868, Z -8.0000, A 0.000, B 0.000, C 0.000 }
gfCNCPoint6[3929] = {X 60.5122, Y 8.2871, Z -8.0000, A 0.000, B 0.000, C 0.000 }
gfCNCPoint6[3930] = {X 61.3577, Y 8.5829, Z -8.0000, A 0.000, B 0.000, C 0.000 }
gfCNCPoint6[3931] = {X 62.1161, Y 9.0595, Z -8.0000, A 0.000, B 0.000, C 0.000 }
gfCNCPoint6[3932] = {X 62.7495, Y 9.6929, Z -8.0000, A 0.000, B 0.000, C 0.000 }
gfCNCPoint6[3933] = {X 63.2260, Y 10.4513, Z -8.0000, A 0.000, B 0.000, C 0.000 }
gfCNCPoint6[3934] = {X 63.5218, Y 11.2967, Z -8.0000, A 0.000, B 0.000, C 0.000 }
gfCNCPoint6[3935] = {X 63.6221, Y 12.1868, Z -8.0000, A 0.000, B 0.000, C 0.000 }
gfCNCPoint6[3936] = {X 63.6219, Y 13.0192, Z -8.0000, A 0.000, B 0.000, C 0.000 }
gfCNCPoint6[3937] = {X 63.5278, Y 13.8416, Z -8.0000, A 0.000, B 0.000, C 0.000 }
gfCNCPoint6[3938] = {X 63.2664, Y 14.6271, Z -8.0000, A 0.000, B 0.000, C 0.000 }
gfCNCPoint6[3939] = {X 62.8489, Y 15.3419, Z -8.0000, A 0.000, B 0.000, C 0.000 }
gfCNCPoint6[3940] = {X 63.1278, Y 16.0764, Z -8.0000, A 0.000, B 0.000, C 0.000 }
gfCNCPoint6[3941] = {X 65.9404, Y 23.5419, Z -8.0000, A 0.000, B 0.000, C 0.000 }
gfCNCPoint6[3942] = {X 71.9123, Y 39.6152, Z -8.0000, A 0.000, B 0.000, C 0.000 }
gfCNCPoint6[3943] = {X 72.2607, Y 40.4916, Z -8.0000, A 0.000, B 0.000, C 0.000 }
gfCNCPoint6[3944] = {X 72.2711, Y 40.5075, Z -8.0000, A 0.000, B 0.000, C 0.000 }
gfCNCPoint6[3945] = {X 72.2868, Y 40.5181, Z -8.0000, A 0.000, B 0.000, C 0.000 }
gfCNCPoint6[3946] = {X 72.3497, Y 40.5450, Z -8.0000, A 0.000, B 0.000, C 0.000 }
gfCNCPoint6[3947] = {X 72.4122, Y 40.5731, Z -8.0000, A 0.000, B 0.000, C 0.000 }
gfCNCPoint6[3948] = {X 73.1913, Y 41.0445, Z -8.0000, A 0.000, B 0.000, C 0.000 }
gfCNCPoint6[3949] = {X 73.8436, Y 41.6799, Z -8.0000, A 0.000, B 0.000, C 0.000 }
gfCNCPoint6[3950] = {X 74.3353, Y 42.4464, Z -8.0000, A 0.000, B 0.000, C 0.000 }
gfCNCPoint6[3951] = {X 74.6408, Y 43.3042, Z -8.0000, A 0.000, B 0.000, C 0.000 }
gfCNCPoint6[3952] = {X 74.7445, Y 44.2089, Z -8.0000, A 0.000, B 0.000, C 0.000 }
gfCNCPoint6[3953] = {X 74.7445, Y 45.0000, Z -8.0000, A 0.000, B 0.000, C 0.000 }
gfCNCPoint6[3954] = {X 74.6442, Y 45.8901, Z -8.0000, A 0.000, B 0.000, C 0.000 }
gfCNCPoint6[3955] = {X 74.3483, Y 46.7355, Z -8.0000, A 0.000, B 0.000, C 0.000 }
gfCNCPoint6[3956] = {X 73.8718, Y 47.4940, Z -8.0000, A 0.000, B 0.000, C 0.000 }
gfCNCPoint6[3957] = {X 73.2384, Y 48.1273, Z -8.0000, A 0.000, B 0.000, C 0.000 }
gfCNCPoint6[3958] = {X 72.4800, Y 48.6039, Z -8.0000, A 0.000, B 0.000, C 0.000 }
gfCNCPoint6[3959] = {X 71.6345, Y 48.8997, Z -8.0000, A 0.000, B 0.000, C 0.000 }
gfCNCPoint6[3960] = {X 70.7445, Y 49.0000, Z -8.0000, A 0.000, B 0.000, C 0.000 }
gfCNCPoint6[3961] = {X 64.1851, Y 49.0000, Z -8.0000, A 0.000, B 0.000, C 0.000 }
gfCNCPoint6[3962] = {X 63.2951, Y 48.8997, Z -8.0000, A 0.000, B 0.000, C 0.000 }
gfCNCPoint6[3963] = {X 62.4496, Y 48.6039, Z -8.0000, A 0.000, B 0.000, C 0.000 }
gfCNCPoint6[3964] = {X 61.6912, Y 48.1273, Z -8.0000, A 0.000, B 0.000, C 0.000 }
gfCNCPoint6[3965] = {X 61.0578, Y 47.4940, Z -8.0000, A 0.000, B 0.000, C 0.000 }
gfCNCPoint6[3966] = {X 60.5813, Y 46.7355, Z -8.0000, A 0.000, B 0.000, C 0.000 }
gfCNCPoint6[3967] = {X 60.2854, Y 45.8901, Z -8.0000, A 0.000, B 0.000, C 0.000 }
gfCNCPoint6[3968] = {X 60.1851, Y 45.0000, Z -8.0000, A 0.000, B 0.000, C 0.000 }
gfCNCPoint6[3969] = {X 60.1855, Y 44.1538, Z -8.0000, A 0.000, B 0.000, C 0.000 }
gfCNCPoint6[3970] = {X 60.2746, Y 43.3674, Z -8.0000, A 0.000, B 0.000, C 0.000 }
gfCNCPoint6[3971] = {X 60.5168, Y 42.6140, Z -8.0000, A 0.000, B 0.000, C 0.000 }
gfCNCPoint6[3972] = {X 60.9025, Y 41.9231, Z -8.0000, A 0.000, B 0.000, C 0.000 }
gfCNCPoint6[3973] = {X 60.9788, Y 41.8179, Z -8.0000, A 0.000, B 0.000, C 0.000 }
gfCNCPoint6[3974] = {X 60.2301, Y 39.7692, Z -8.0000, A 0.000, B 0.000, C 0.000 }
gfCNCPoint6[3975] = {X 51.8432, Y 39.7692, Z -8.0000, A 0.000, B 0.000, C 0.000 }
gfCNCPoint6[3976] = {X 51.8432, Y 39.8040, Z -8.0000, A 0.000, B 0.000, C 0.000 }
gfCNCPoint6[3977] = {X 50.9823, Y 42.1173, Z -8.0000, A 0.000, B 0.000, C 0.000 }
gfCNCPoint6[3978] = {X 51.0732, Y 42.2728, Z -8.0000, A 0.000, B 0.000, C 0.000 }
gfCNCPoint6[3979] = {X 51.3482, Y 42.8869, Z -8.0000, A 0.000, B 0.000, C 0.000 }
gfCNCPoint6[3980] = {X 51.5164, Y 43.5384, Z -8.0000, A 0.000, B 0.000, C 0.000 }
gfCNCPoint6[3981] = {X 51.5729, Y 44.2089, Z -8.0000, A 0.000, B 0.000, C 0.000 }
gfCNCPoint6[3982] = {X 51.5729, Y 45.0000, Z -8.0000, A 0.000, B 0.000, C 0.000 }
gfCNCPoint6[3983] = {X 51.4726, Y 45.8901, Z -8.0000, A 0.000, B 0.000, C 0.000 }
gfCNCPoint6[3984] = {X 51.1768, Y 46.7355, Z -8.0000, A 0.000, B 0.000, C 0.000 }
gfCNCPoint6[3985] = {X 50.7003, Y 47.4940, Z -8.0000, A 0.000, B 0.000, C 0.000 }
gfCNCPoint6[3986] = {X 50.0669, Y 48.1273, Z -8.0000, A 0.000, B 0.000, C 0.000 }
gfCNCPoint6[3987] = {X 49.3085, Y 48.6039, Z -8.0000, A 0.000, B 0.000, C 0.000 }
gfCNCPoint6[3988] = {X 48.4630, Y 48.8997, Z -8.0000, A 0.000, B 0.000, C 0.000 }
gfCNCPoint6[3989] = {X 47.5729, Y 49.0000, Z -8.0000, A 0.000, B 0.000, C 0.000 }
gfCNCPoint6[3990] = {X 40.6393, Y 49.0000, Z -8.0000, A 0.000, B 0.000, C 0.000 }
gfCNCPoint6[3991] = {X 39.7492, Y 48.8997, Z -8.0000, A 0.000, B 0.000, C 0.000 }
gfCNCPoint6[3992] = {X 38.9038, Y 48.6039, Z -8.0000, A 0.000, B 0.000, C 0.000 }
gfCNCPoint6[3993] = {X 38.1453, Y 48.1273, Z -8.0000, A 0.000, B 0.000, C 0.000 }
gfCNCPoint6[3994] = {X 37.5120, Y 47.4940, Z -8.0000, A 0.000, B 0.000, C 0.000 }
gfCNCPoint6[3995] = {X 37.0354, Y 46.7355, Z -8.0000, A 0.000, B 0.000, C 0.000 }
gfCNCPoint6[3996] = {X 36.7396, Y 45.8901, Z -8.0000, A 0.000, B 0.000, C 0.000 }
gfCNCPoint6[3997] = {X 36.6393, Y 45.0000, Z -8.0000, A 0.000, B 0.000, C 0.000 }
gfCNCPoint6[3998] = {X 36.6397, Y 44.1538, Z -8.0000, A 0.000, B 0.000, C 0.000 }
gfCNCPoint6[3999] = {X 36.7563, Y 43.2486, Z -8.0000, A 0.000, B 0.000, C 0.000 }
gfCNCPoint6[4000] = {X 37.0750, Y 42.3933, Z -8.0000, A 0.000, B 0.000, C 0.000 }
gfCNCPoint6[4001] = {X 37.5793, Y 41.6327, Z -8.0000, A 0.000, B 0.000, C 0.000 }
gfCNCPoint6[4002] = {X 38.2429, Y 41.0061, Z -8.0000, A 0.000, B 0.000, C 0.000 }
gfCNCPoint6[4003] = {X 39.0313, Y 40.5462, Z -8.0000, A 0.000, B 0.000, C 0.000 }
gfCNCPoint6[4004] = {X 39.0813, Y 40.5247, Z -8.0000, A 0.000, B 0.000, C 0.000 }
gfCNCPoint6[4005] = {X 39.1315, Y 40.5038, Z -8.0000, A 0.000, B 0.000, C 0.000 }
gfCNCPoint6[4006] = {X 39.1655, Y 40.4817, Z -8.0000, A 0.000, B 0.000, C 0.000 }
gfCNCPoint6[4007] = {X 39.1888, Y 40.4485, Z -8.0000, A 0.000, B 0.000, C 0.000 }
gfCNCPoint6[4008] = {X 39.2125, Y 40.3954, Z -8.0000, A 0.000, B 0.000, C 0.000 }
gfCNCPoint6[4009] = {X 39.2361, Y 40.3422, Z -8.0000, A 0.000, B 0.000, C 0.000 }
gfCNCPoint6[4010] = {X 39.8247, Y 38.9502, Z -8.0000, A 0.000, B 0.000, C 0.000 }
gfCNCPoint6[4011] = {X 40.3639, Y 37.5383, Z -8.0000, A 0.000, B 0.000, C 0.000 }
gfCNCPoint6[4012] = {X 43.9473, Y 27.9191, Z -8.0000, A 0.000, B 0.000, C 0.000 }
gfCNCPoint6[4013] = {X 40.1240, Y 26.4948, Z -8.0000, A 0.000, B 0.000, C 0.000 }
gfCNCPoint6[4014] = {X 40.1240, Y 26.4948, Z -5.0000, A 0.000, B 0.000, C 0.000 }
gfCNCPoint6[4015] = {X 40.1240, Y 26.4948, Z 11.0000, A 0.000, B 0.000, C 0.000 }
gfCNCPoint6[4016] = {X 79.0216, Y 28.5909, Z 11.0000, A 0.000, B 0.000, C 0.000 }
gfCNCPoint6[4017] = {X 79.0216, Y 28.5909, Z -5.0000, A 0.000, B 0.000, C 0.000 }
gfCNCPoint6[4018] = {X 79.0216, Y 28.5909, Z -8.0000, A 0.000, B 0.000, C 0.000 }
gfCNCPoint6[4019] = {X 83.1016, Y 28.5909, Z -8.0000, A 0.000, B 0.000, C 0.000 }
gfCNCPoint6[4020] = {X 83.1017, Y 16.2734, Z -8.0000, A 0.000, B 0.000, C 0.000 }
gfCNCPoint6[4021] = {X 82.4635, Y 15.6023, Z -8.0000, A 0.000, B 0.000, C 0.000 }
gfCNCPoint6[4022] = {X 81.9830, Y 14.8106, Z -8.0000, A 0.000, B 0.000, C 0.000 }
gfCNCPoint6[4023] = {X 81.6823, Y 13.9347, Z -8.0000, A 0.000, B 0.000, C 0.000 }
gfCNCPoint6[4024] = {X 81.5752, Y 13.0148, Z -8.0000, A 0.000, B 0.000, C 0.000 }
gfCNCPoint6[4025] = {X 81.5751, Y 12.1868, Z -8.0000, A 0.000, B 0.000, C 0.000 }
gfCNCPoint6[4026] = {X 81.6834, Y 11.2255, Z -8.0000, A 0.000, B 0.000, C 0.000 }
gfCNCPoint6[4027] = {X 82.0029, Y 10.3124, Z -8.0000, A 0.000, B 0.000, C 0.000 }
gfCNCPoint6[4028] = {X 82.5176, Y 9.4933, Z -8.0000, A 0.000, B 0.000, C 0.000 }
gfCNCPoint6[4029] = {X 83.2016, Y 8.8093, Z -8.0000, A 0.000, B 0.000, C 0.000 }
gfCNCPoint6[4030] = {X 84.0207, Y 8.2946, Z -8.0000, A 0.000, B 0.000, C 0.000 }
gfCNCPoint6[4031] = {X 84.9338, Y 7.9751, Z -8.0000, A 0.000, B 0.000, C 0.000 }
gfCNCPoint6[4032] = {X 85.8951, Y 7.8668, Z -8.0000, A 0.000, B 0.000, C 0.000 }
gfCNCPoint6[4033] = {X 94.0497, Y 7.8668, Z -8.0000, A 0.000, B 0.000, C 0.000 }
gfCNCPoint6[4034] = {X 95.0110, Y 7.9751, Z -8.0000, A 0.000, B 0.000, C 0.000 }
gfCNCPoint6[4035] = {X 95.9240, Y 8.2946, Z -8.0000, A 0.000, B 0.000, C 0.000 }
gfCNCPoint6[4036] = {X 96.7431, Y 8.8093, Z -8.0000, A 0.000, B 0.000, C 0.000 }
gfCNCPoint6[4037] = {X 97.4272, Y 9.4933, Z -8.0000, A 0.000, B 0.000, C 0.000 }
gfCNCPoint6[4038] = {X 97.9419, Y 10.3124, Z -8.0000, A 0.000, B 0.000, C 0.000 }
gfCNCPoint6[4039] = {X 98.2614, Y 11.2255, Z -8.0000, A 0.000, B 0.000, C 0.000 }
gfCNCPoint6[4040] = {X 98.3697, Y 12.1868, Z -8.0000, A 0.000, B 0.000, C 0.000 }
gfCNCPoint6[4041] = {X 98.3697, Y 12.9782, Z -8.0000, A 0.000, B 0.000, C 0.000 }
gfCNCPoint6[4042] = {X 98.2968, Y 13.7675, Z -8.0000, A 0.000, B 0.000, C 0.000 }
gfCNCPoint6[4043] = {X 98.0809, Y 14.5303, Z -8.0000, A 0.000, B 0.000, C 0.000 }
gfCNCPoint6[4044] = {X 97.7293, Y 15.2407, Z -8.0000, A 0.000, B 0.000, C 0.000 }
gfCNCPoint6[4045] = {X 101.8771, Y 25.5237, Z -8.0000, A 0.000, B 0.000, C 0.000 }
gfCNCPoint6[4046] = {X 106.0160, Y 15.2206, Z -8.0000, A 0.000, B 0.000, C 0.000 }
gfCNCPoint6[4047] = {X 105.6759, Y 14.5280, Z -8.0000, A 0.000, B 0.000, C 0.000 }
gfCNCPoint6[4048] = {X 105.4645, Y 13.7858, Z -8.0000, A 0.000, B 0.000, C 0.000 }
gfCNCPoint6[4049] = {X 105.3885, Y 13.0179, Z -8.0000, A 0.000, B 0.000, C 0.000 }
gfCNCPoint6[4050] = {X 105.3883, Y 12.1868, Z -8.0000, A 0.000, B 0.000, C 0.000 }
gfCNCPoint6[4051] = {X 105.4966, Y 11.2255, Z -8.0000, A 0.000, B 0.000, C 0.000 }
gfCNCPoint6[4052] = {X 105.8161, Y 10.3124, Z -8.0000, A 0.000, B 0.000, C 0.000 }
gfCNCPoint6[4053] = {X 106.3308, Y 9.4933, Z -8.0000, A 0.000, B 0.000, C 0.000 }
gfCNCPoint6[4054] = {X 107.0148, Y 8.8093, Z -8.0000, A 0.000, B 0.000, C 0.000 }
gfCNCPoint6[4055] = {X 107.8339, Y 8.2946, Z -8.0000, A 0.000, B 0.000, C 0.000 }
gfCNCPoint6[4056] = {X 108.7470, Y 7.9751, Z -8.0000, A 0.000, B 0.000, C 0.000 }
gfCNCPoint6[4057] = {X 109.7083, Y 7.8668, Z -8.0000, A 0.000, B 0.000, C 0.000 }
gfCNCPoint6[4058] = {X 117.7916, Y 7.8668, Z -8.0000, A 0.000, B 0.000, C 0.000 }
gfCNCPoint6[4059] = {X 118.7529, Y 7.9751, Z -8.0000, A 0.000, B 0.000, C 0.000 }
gfCNCPoint6[4060] = {X 119.6660, Y 8.2946, Z -8.0000, A 0.000, B 0.000, C 0.000 }
gfCNCPoint6[4061] = {X 120.4851, Y 8.8093, Z -8.0000, A 0.000, B 0.000, C 0.000 }
gfCNCPoint6[4062] = {X 121.1691, Y 9.4933, Z -8.0000, A 0.000, B 0.000, C 0.000 }
gfCNCPoint6[4063] = {X 121.6838, Y 10.3124, Z -8.0000, A 0.000, B 0.000, C 0.000 }
gfCNCPoint6[4064] = {X 122.0033, Y 11.2255, Z -8.0000, A 0.000, B 0.000, C 0.000 }
gfCNCPoint6[4065] = {X 122.1116, Y 12.1868, Z -8.0000, A 0.000, B 0.000, C 0.000 }
gfCNCPoint6[4066] = {X 122.1116, Y 12.9782, Z -8.0000, A 0.000, B 0.000, C 0.000 }
gfCNCPoint6[4067] = {X 122.0103, Y 13.9078, Z -8.0000, A 0.000, B 0.000, C 0.000 }
gfCNCPoint6[4068] = {X 121.7114, Y 14.7939, Z -8.0000, A 0.000, B 0.000, C 0.000 }
gfCNCPoint6[4069] = {X 121.2288, Y 15.5949, Z -8.0000, A 0.000, B 0.000, C 0.000 }
gfCNCPoint6[4070] = {X 120.5851, Y 16.2732, Z -8.0000, A 0.000, B 0.000, C 0.000 }
gfCNCPoint6[4071] = {X 120.5853, Y 40.9148, Z -8.0000, A 0.000, B 0.000, C 0.000 }
gfCNCPoint6[4072] = {X 120.6230, Y 40.9460, Z -8.0000, A 0.000, B 0.000, C 0.000 }
gfCNCPoint6[4073] = {X 121.2460, Y 41.6147, Z -8.0000, A 0.000, B 0.000, C 0.000 }
gfCNCPoint6[4074] = {X 121.7145, Y 42.3996, Z -8.0000, A 0.000, B 0.000, C 0.000 }
gfCNCPoint6[4075] = {X 122.0073, Y 43.2654, Z -8.0000, A 0.000, B 0.000, C 0.000 }
gfCNCPoint6[4076] = {X 122.1114, Y 44.1734, Z -8.0000, A 0.000, B 0.000, C 0.000 }
gfCNCPoint6[4077] = {X 122.1116, Y 45.0000, Z -8.0000, A 0.000, B 0.000, C 0.000 }
gfCNCPoint6[4078] = {X 122.0033, Y 45.9613, Z -8.0000, A 0.000, B 0.000, C 0.000 }
gfCNCPoint6[4079] = {X 121.6838, Y 46.8744, Z -8.0000, A 0.000, B 0.000, C 0.000 }
gfCNCPoint6[4080] = {X 121.1691, Y 47.6935, Z -8.0000, A 0.000, B 0.000, C 0.000 }
gfCNCPoint6[4081] = {X 120.4851, Y 48.3775, Z -8.0000, A 0.000, B 0.000, C 0.000 }
gfCNCPoint6[4082] = {X 119.6660, Y 48.8922, Z -8.0000, A 0.000, B 0.000, C 0.000 }
gfCNCPoint6[4083] = {X 118.7529, Y 49.2117, Z -8.0000, A 0.000, B 0.000, C 0.000 }
gfCNCPoint6[4084] = {X 117.7916, Y 49.3200, Z -8.0000, A 0.000, B 0.000, C 0.000 }
gfCNCPoint6[4085] = {X 111.9185, Y 49.3200, Z -8.0000, A 0.000, B 0.000, C 0.000 }
gfCNCPoint6[4086] = {X 110.9619, Y 49.2128, Z -8.0000, A 0.000, B 0.000, C 0.000 }
gfCNCPoint6[4087] = {X 110.0529, Y 48.8964, Z -8.0000, A 0.000, B 0.000, C 0.000 }
gfCNCPoint6[4088] = {X 109.2365, Y 48.3866, Z -8.0000, A 0.000, B 0.000, C 0.000 }
gfCNCPoint6[4089] = {X 108.5532, Y 47.7087, Z -8.0000, A 0.000, B 0.000, C 0.000 }
gfCNCPoint6[4090] = {X 108.0369, Y 46.8963, Z -8.0000, A 0.000, B 0.000, C 0.000 }
gfCNCPoint6[4091] = {X 107.7134, Y 45.9898, Z -8.0000, A 0.000, B 0.000, C 0.000 }
gfCNCPoint6[4092] = {X 107.5986, Y 45.0341, Z -8.0000, A 0.000, B 0.000, C 0.000 }
gfCNCPoint6[4093] = {X 107.5985, Y 44.1753, Z -8.0000, A 0.000, B 0.000, C 0.000 }
gfCNCPoint6[4094] = {X 107.6336, Y 43.6370, Z -8.0000, A 0.000, B 0.000, C 0.000 }
gfCNCPoint6[4095] = {X 107.7382, Y 43.1079, Z -8.0000, A 0.000, B 0.000, C 0.000 }
gfCNCPoint6[4096] = {X 107.9074, Y 42.6045, Z -8.0000, A 0.000, B 0.000, C 0.000 }
gfCNCPoint6[4097] = {X 108.1396, Y 42.1269, Z -8.0000, A 0.000, B 0.000, C 0.000 }
gfCNCPoint6[4098] = {X 108.5884, Y 41.4606, Z -8.0000, A 0.000, B 0.000, C 0.000 }
gfCNCPoint6[4099] = {X 109.1246, Y 40.8623, Z -8.0000, A 0.000, B 0.000, C 0.000 }
gfCNCPoint6[4100] = {X 109.1245, Y 39.2994, Z -8.0000, A 0.000, B 0.000, C 0.000 }
gfCNCPoint6[4101] = {X 106.1118, Y 46.6615, Z -8.0000, A 0.000, B 0.000, C 0.000 }
gfCNCPoint6[4102] = {X 105.7417, Y 47.3611, Z -8.0000, A 0.000, B 0.000, C 0.000 }
gfCNCPoint6[4103] = {X 105.2502, Y 47.9815, Z -8.0000, A 0.000, B 0.000, C 0.000 }
gfCNCPoint6[4104] = {X 104.6538, Y 48.5018, Z -8.0000, A 0.000, B 0.000, C 0.000 }
gfCNCPoint6[4105] = {X 103.9724, Y 48.9046, Z -8.0000, A 0.000, B 0.000, C 0.000 }
gfCNCPoint6[4106] = {X 103.0287, Y 49.2242, Z -8.0000, A 0.000, B 0.000, C 0.000 }
gfCNCPoint6[4107] = {X 102.0368, Y 49.3191, Z -8.0000, A 0.000, B 0.000, C 0.000 }
gfCNCPoint6[4108] = {X 101.0496, Y 49.1842, Z -8.0000, A 0.000, B 0.000, C 0.000 }
gfCNCPoint6[4109] = {X 100.1195, Y 48.8268, Z -8.0000, A 0.000, B 0.000, C 0.000 }
gfCNCPoint6[4110] = {X 99.2961, Y 48.2657, Z -8.0000, A 0.000, B 0.000, C 0.000 }
gfCNCPoint6[4111] = {X 98.6231, Y 47.5309, Z -8.0000, A 0.000, B 0.000, C 0.000 }
gfCNCPoint6[4112] = {X 98.1363, Y 46.6615, Z -8.0000, A 0.000, B 0.000, C 0.000 }
gfCNCPoint6[4113] = {X 95.1323, Y 39.3148, Z -8.0000, A 0.000, B 0.000, C 0.000 }
gfCNCPoint6[4114] = {X 95.1324, Y 40.9045, Z -8.0000, A 0.000, B 0.000, C 0.000 }
gfCNCPoint6[4115] = {X 95.6566, Y 41.4409, Z -8.0000, A 0.000, B 0.000, C 0.000 }
gfCNCPoint6[4116] = {X 96.0820, Y 42.0586, Z -8.0000, A 0.000, B 0.000, C 0.000 }
gfCNCPoint6[4117] = {X 96.3315, Y 42.5710, Z -8.0000, A 0.000, B 0.000, C 0.000 }
gfCNCPoint6[4118] = {X 96.5125, Y 43.1114, Z -8.0000, A 0.000, B 0.000, C 0.000 }
gfCNCPoint6[4119] = {X 96.6201, Y 43.6545, Z -8.0000, A 0.000, B 0.000, C 0.000 }
gfCNCPoint6[4120] = {X 96.6585, Y 44.2067, Z -8.0000, A 0.000, B 0.000, C 0.000 }
gfCNCPoint6[4121] = {X 96.6583, Y 45.0415, Z -8.0000, A 0.000, B 0.000, C 0.000 }
gfCNCPoint6[4122] = {X 96.5422, Y 45.9960, Z -8.0000, A 0.000, B 0.000, C 0.000 }
gfCNCPoint6[4123] = {X 96.2178, Y 46.9011, Z -8.0000, A 0.000, B 0.000, C 0.000 }
gfCNCPoint6[4124] = {X 95.7012, Y 47.7120, Z -8.0000, A 0.000, B 0.000, C 0.000 }
gfCNCPoint6[4125] = {X 95.0181, Y 48.3886, Z -8.0000, A 0.000, B 0.000, C 0.000 }
gfCNCPoint6[4126] = {X 94.2022, Y 48.8973, Z -8.0000, A 0.000, B 0.000, C 0.000 }
gfCNCPoint6[4127] = {X 93.2940, Y 49.2130, Z -8.0000, A 0.000, B 0.000, C 0.000 }
gfCNCPoint6[4128] = {X 92.3385, Y 49.3200, Z -8.0000, A 0.000, B 0.000, C 0.000 }
gfCNCPoint6[4129] = {X 85.8951, Y 49.3200, Z -8.0000, A 0.000, B 0.000, C 0.000 }
gfCNCPoint6[4130] = {X 84.9387, Y 49.2128, Z -8.0000, A 0.000, B 0.000, C 0.000 }
gfCNCPoint6[4131] = {X 84.0297, Y 48.8965, Z -8.0000, A 0.000, B 0.000, C 0.000 }
gfCNCPoint6[4132] = {X 83.2134, Y 48.3869, Z -8.0000, A 0.000, B 0.000, C 0.000 }
gfCNCPoint6[4133] = {X 82.5301, Y 47.7091, Z -8.0000, A 0.000, B 0.000, C 0.000 }
gfCNCPoint6[4134] = {X 82.0138, Y 46.8970, Z -8.0000, A 0.000, B 0.000, C 0.000 }
gfCNCPoint6[4135] = {X 81.6902, Y 45.9906, Z -8.0000, A 0.000, B 0.000, C 0.000 }
gfCNCPoint6[4136] = {X 81.5752, Y 45.0351, Z -8.0000, A 0.000, B 0.000, C 0.000 }
gfCNCPoint6[4137] = {X 81.5751, Y 44.2073, Z -8.0000, A 0.000, B 0.000, C 0.000 }
gfCNCPoint6[4138] = {X 81.6796, Y 43.2778, Z -8.0000, A 0.000, B 0.000, C 0.000 }
gfCNCPoint6[4139] = {X 81.9793, Y 42.3918, Z -8.0000, A 0.000, B 0.000, C 0.000 }
gfCNCPoint6[4140] = {X 82.4607, Y 41.5897, Z -8.0000, A 0.000, B 0.000, C 0.000 }
gfCNCPoint6[4141] = {X 83.1016, Y 40.9085, Z -8.0000, A 0.000, B 0.000, C 0.000 }
gfCNCPoint6[4142] = {X 83.1016, Y 28.5909, Z -8.0000, A 0.000, B 0.000, C 0.000 }
gfCNCPoint6[4143] = {X 79.1016, Y 28.5909, Z -8.0000, A 0.000, B 0.000, C 0.000 }
gfCNCPoint6[4144] = {X 83.1816, Y 28.5909, Z -8.0000, A 0.000, B 0.000, C 0.000 }
gfCNCPoint6[4145] = {X 83.1817, Y 16.2361, Z -8.0000, A 0.000, B 0.000, C 0.000 }
gfCNCPoint6[4146] = {X 82.5439, Y 15.5756, Z -8.0000, A 0.000, B 0.000, C 0.000 }
gfCNCPoint6[4147] = {X 82.0633, Y 14.7934, Z -8.0000, A 0.000, B 0.000, C 0.000 }
gfCNCPoint6[4148] = {X 81.7624, Y 13.9260, Z -8.0000, A 0.000, B 0.000, C 0.000 }
gfCNCPoint6[4149] = {X 81.6552, Y 13.0142, Z -8.0000, A 0.000, B 0.000, C 0.000 }
gfCNCPoint6[4150] = {X 81.6551, Y 12.1868, Z -8.0000, A 0.000, B 0.000, C 0.000 }
gfCNCPoint6[4151] = {X 81.7614, Y 11.2433, Z -8.0000, A 0.000, B 0.000, C 0.000 }
gfCNCPoint6[4152] = {X 82.0750, Y 10.3472, Z -8.0000, A 0.000, B 0.000, C 0.000 }
gfCNCPoint6[4153] = {X 82.5801, Y 9.5432, Z -8.0000, A 0.000, B 0.000, C 0.000 }
gfCNCPoint6[4154] = {X 83.2515, Y 8.8719, Z -8.0000, A 0.000, B 0.000, C 0.000 }
gfCNCPoint6[4155] = {X 84.0554, Y 8.3667, Z -8.0000, A 0.000, B 0.000, C 0.000 }
gfCNCPoint6[4156] = {X 84.9516, Y 8.0531, Z -8.0000, A 0.000, B 0.000, C 0.000 }
gfCNCPoint6[4157] = {X 85.8951, Y 7.9468, Z -8.0000, A 0.000, B 0.000, C 0.000 }
gfCNCPoint6[4158] = {X 94.0497, Y 7.9468, Z -8.0000, A 0.000, B 0.000, C 0.000 }
gfCNCPoint6[4159] = {X 94.9932, Y 8.0531, Z -8.0000, A 0.000, B 0.000, C 0.000 }
gfCNCPoint6[4160] = {X 95.8893, Y 8.3667, Z -8.0000, A 0.000, B 0.000, C 0.000 }
gfCNCPoint6[4161] = {X 96.6933, Y 8.8718, Z -8.0000, A 0.000, B 0.000, C 0.000 }
gfCNCPoint6[4162] = {X 97.3646, Y 9.5432, Z -8.0000, A 0.000, B 0.000, C 0.000 }
gfCNCPoint6[4163] = {X 97.8698, Y 10.3471, Z -8.0000, A 0.000, B 0.000, C 0.000 }
gfCNCPoint6[4164] = {X 98.1834, Y 11.2433, Z -8.0000, A 0.000, B 0.000, C 0.000 }
gfCNCPoint6[4165] = {X 98.2897, Y 12.1868, Z -8.0000, A 0.000, B 0.000, C 0.000 }
gfCNCPoint6[4166] = {X 98.2897, Y 12.9782, Z -8.0000, A 0.000, B 0.000, C 0.000 }
gfCNCPoint6[4167] = {X 98.2156, Y 13.7661, Z -8.0000, A 0.000, B 0.000, C 0.000 }
gfCNCPoint6[4168] = {X 97.9965, Y 14.5265, Z -8.0000, A 0.000, B 0.000, C 0.000 }
gfCNCPoint6[4169] = {X 97.6399, Y 15.2330, Z -8.0000, A 0.000, B 0.000, C 0.000 }
gfCNCPoint6[4170] = {X 101.8772, Y 25.7379, Z -8.0000, A 0.000, B 0.000, C 0.000 }
gfCNCPoint6[4171] = {X 106.1052, Y 15.2131, Z -8.0000, A 0.000, B 0.000, C 0.000 }
gfCNCPoint6[4172] = {X 105.7602, Y 14.5240, Z -8.0000, A 0.000, B 0.000, C 0.000 }
gfCNCPoint6[4173] = {X 105.5456, Y 13.7839, Z -8.0000, A 0.000, B 0.000, C 0.000 }
gfCNCPoint6[4174] = {X 105.4685, Y 13.0172, Z -8.0000, A 0.000, B 0.000, C 0.000 }
gfCNCPoint6[4175] = {X 105.4683, Y 12.1868, Z -8.0000, A 0.000, B 0.000, C 0.000 }
gfCNCPoint6[4176] = {X 105.5746, Y 11.2433, Z -8.0000, A 0.000, B 0.000, C 0.000 }
gfCNCPoint6[4177] = {X 105.8882, Y 10.3471, Z -8.0000, A 0.000, B 0.000, C 0.000 }
gfCNCPoint6[4178] = {X 106.3933, Y 9.5432, Z -8.0000, A 0.000, B 0.000, C 0.000 }
gfCNCPoint6[4179] = {X 107.0647, Y 8.8718, Z -8.0000, A 0.000, B 0.000, C 0.000 }
gfCNCPoint6[4180] = {X 107.8686, Y 8.3667, Z -8.0000, A 0.000, B 0.000, C 0.000 }
gfCNCPoint6[4181] = {X 108.7648, Y 8.0531, Z -8.0000, A 0.000, B 0.000, C 0.000 }
gfCNCPoint6[4182] = {X 109.7083, Y 7.9468, Z -8.0000, A 0.000, B 0.000, C 0.000 }
gfCNCPoint6[4183] = {X 117.7916, Y 7.9468, Z -8.0000, A 0.000, B 0.000, C 0.000 }
gfCNCPoint6[4184] = {X 118.7351, Y 8.0531, Z -8.0000, A 0.000, B 0.000, C 0.000 }
gfCNCPoint6[4185] = {X 119.6312, Y 8.3667, Z -8.0000, A 0.000, B 0.000, C 0.000 }
gfCNCPoint6[4186] = {X 120.4352, Y 8.8718, Z -8.0000, A 0.000, B 0.000, C 0.000 }
gfCNCPoint6[4187] = {X 121.1065, Y 9.5432, Z -8.0000, A 0.000, B 0.000, C 0.000 }
gfCNCPoint6[4188] = {X 121.6117, Y 10.3471, Z -8.0000, A 0.000, B 0.000, C 0.000 }
gfCNCPoint6[4189] = {X 121.9253, Y 11.2433, Z -8.0000, A 0.000, B 0.000, C 0.000 }
gfCNCPoint6[4190] = {X 122.0316, Y 12.1868, Z -8.0000, A 0.000, B 0.000, C 0.000 }
gfCNCPoint6[4191] = {X 122.0316, Y 12.9782, Z -8.0000, A 0.000, B 0.000, C 0.000 }
gfCNCPoint6[4192] = {X 121.9302, Y 13.8996, Z -8.0000, A 0.000, B 0.000, C 0.000 }
gfCNCPoint6[4193] = {X 121.6310, Y 14.7770, Z -8.0000, A 0.000, B 0.000, C 0.000 }
gfCNCPoint6[4194] = {X 121.1483, Y 15.5684, Z -8.0000, A 0.000, B 0.000, C 0.000 }
gfCNCPoint6[4195] = {X 120.5051, Y 16.2360, Z -8.0000, A 0.000, B 0.000, C 0.000 }
gfCNCPoint6[4196] = {X 120.5053, Y 40.9524, Z -8.0000, A 0.000, B 0.000, C 0.000 }
gfCNCPoint6[4197] = {X 120.5712, Y 41.0071, Z -8.0000, A 0.000, B 0.000, C 0.000 }
gfCNCPoint6[4198] = {X 121.1825, Y 41.6633, Z -8.0000, A 0.000, B 0.000, C 0.000 }
gfCNCPoint6[4199] = {X 121.6420, Y 42.4335, Z -8.0000, A 0.000, B 0.000, C 0.000 }
gfCNCPoint6[4200] = {X 121.9293, Y 43.2831, Z -8.0000, A 0.000, B 0.000, C 0.000 }
gfCNCPoint6[4201] = {X 122.0314, Y 44.1740, Z -8.0000, A 0.000, B 0.000, C 0.000 }
gfCNCPoint6[4202] = {X 122.0316, Y 45.0000, Z -8.0000, A 0.000, B 0.000, C 0.000 }
gfCNCPoint6[4203] = {X 121.9253, Y 45.9435, Z -8.0000, A 0.000, B 0.000, C 0.000 }
gfCNCPoint6[4204] = {X 121.6117, Y 46.8397, Z -8.0000, A 0.000, B 0.000, C 0.000 }
gfCNCPoint6[4205] = {X 121.1065, Y 47.6436, Z -8.0000, A 0.000, B 0.000, C 0.000 }
gfCNCPoint6[4206] = {X 120.4352, Y 48.3150, Z -8.0000, A 0.000, B 0.000, C 0.000 }
gfCNCPoint6[4207] = {X 119.6312, Y 48.8201, Z -8.0000, A 0.000, B 0.000, C 0.000 }
gfCNCPoint6[4208] = {X 118.7351, Y 49.1337, Z -8.0000, A 0.000, B 0.000, C 0.000 }
gfCNCPoint6[4209] = {X 117.7916, Y 49.2400, Z -8.0000, A 0.000, B 0.000, C 0.000 }
gfCNCPoint6[4210] = {X 111.9185, Y 49.2400, Z -8.0000, A 0.000, B 0.000, C 0.000 }
gfCNCPoint6[4211] = {X 110.9797, Y 49.1348, Z -8.0000, A 0.000, B 0.000, C 0.000 }
gfCNCPoint6[4212] = {X 110.0874, Y 48.8242, Z -8.0000, A 0.000, B 0.000, C 0.000 }
gfCNCPoint6[4213] = {X 109.2861, Y 48.3239, Z -8.0000, A 0.000, B 0.000, C 0.000 }
gfCNCPoint6[4214] = {X 108.6155, Y 47.6585, Z -8.0000, A 0.000, B 0.000, C 0.000 }
gfCNCPoint6[4215] = {X 108.1088, Y 46.8612, Z -8.0000, A 0.000, B 0.000, C 0.000 }
gfCNCPoint6[4216] = {X 107.7913, Y 45.9714, Z -8.0000, A 0.000, B 0.000, C 0.000 }
gfCNCPoint6[4217] = {X 107.6786, Y 45.0335, Z -8.0000, A 0.000, B 0.000, C 0.000 }
gfCNCPoint6[4218] = {X 107.6785, Y 44.1753, Z -8.0000, A 0.000, B 0.000, C 0.000 }
gfCNCPoint6[4219] = {X 107.7129, Y 43.6474, Z -8.0000, A 0.000, B 0.000, C 0.000 }
gfCNCPoint6[4220] = {X 107.8155, Y 43.1285, Z -8.0000, A 0.000, B 0.000, C 0.000 }
gfCNCPoint6[4221] = {X 107.9815, Y 42.6348, Z -8.0000, A 0.000, B 0.000, C 0.000 }
gfCNCPoint6[4222] = {X 108.2092, Y 42.1664, Z -8.0000, A 0.000, B 0.000, C 0.000 }
gfCNCPoint6[4223] = {X 108.6620, Y 41.4962, Z -8.0000, A 0.000, B 0.000, C 0.000 }
gfCNCPoint6[4224] = {X 109.2046, Y 40.8963, Z -8.0000, A 0.000, B 0.000, C 0.000 }
gfCNCPoint6[4225] = {X 109.2045, Y 39.1629, Z -8.0000, A 0.000, B 0.000, C 0.000 }
gfCNCPoint6[4226] = {X 109.0939, Y 39.1629, Z -8.0000, A 0.000, B 0.000, C 0.000 }
gfCNCPoint6[4227] = {X 106.0379, Y 46.6307, Z -8.0000, A 0.000, B 0.000, C 0.000 }
gfCNCPoint6[4228] = {X 105.6747, Y 47.3174, Z -8.0000, A 0.000, B 0.000, C 0.000 }
gfCNCPoint6[4229] = {X 105.1923, Y 47.9263, Z -8.0000, A 0.000, B 0.000, C 0.000 }
gfCNCPoint6[4230] = {X 104.6069, Y 48.4370, Z -8.0000, A 0.000, B 0.000, C 0.000 }
gfCNCPoint6[4231] = {X 103.9382, Y 48.8323, Z -8.0000, A 0.000, B 0.000, C 0.000 }
gfCNCPoint6[4232] = {X 103.0119, Y 49.1460, Z -8.0000, A 0.000, B 0.000, C 0.000 }
gfCNCPoint6[4233] = {X 102.0384, Y 49.2391, Z -8.0000, A 0.000, B 0.000, C 0.000 }
gfCNCPoint6[4234] = {X 101.0695, Y 49.1068, Z -8.0000, A 0.000, B 0.000, C 0.000 }
gfCNCPoint6[4235] = {X 100.1566, Y 48.7559, Z -8.0000, A 0.000, B 0.000, C 0.000 }
gfCNCPoint6[4236] = {X 99.3484, Y 48.2052, Z -8.0000, A 0.000, B 0.000, C 0.000 }
gfCNCPoint6[4237] = {X 98.6879, Y 47.4840, Z -8.0000, A 0.000, B 0.000, C 0.000 }
gfCNCPoint6[4238] = {X 98.2102, Y 46.6307, Z -8.0000, A 0.000, B 0.000, C 0.000 }
gfCNCPoint6[4239] = {X 95.0523, Y 38.9078, Z -8.0000, A 0.000, B 0.000, C 0.000 }
gfCNCPoint6[4240] = {X 95.0524, Y 40.9413, Z -8.0000, A 0.000, B 0.000, C 0.000 }
gfCNCPoint6[4241] = {X 95.5832, Y 41.4777, Z -8.0000, A 0.000, B 0.000, C 0.000 }
gfCNCPoint6[4242] = {X 96.0125, Y 42.0982, Z -8.0000, A 0.000, B 0.000, C 0.000 }
gfCNCPoint6[4243] = {X 96.2574, Y 42.6013, Z -8.0000, A 0.000, B 0.000, C 0.000 }
gfCNCPoint6[4244] = {X 96.4352, Y 43.1318, Z -8.0000, A 0.000, B 0.000, C 0.000 }
gfCNCPoint6[4245] = {X 96.5408, Y 43.6650, Z -8.0000, A 0.000, B 0.000, C 0.000 }
gfCNCPoint6[4246] = {X 96.5785, Y 44.2073, Z -8.0000, A 0.000, B 0.000, C 0.000 }
gfCNCPoint6[4247] = {X 96.5783, Y 45.0408, Z -8.0000, A 0.000, B 0.000, C 0.000 }
gfCNCPoint6[4248] = {X 96.4643, Y 45.9775, Z -8.0000, A 0.000, B 0.000, C 0.000 }
gfCNCPoint6[4249] = {X 96.1459, Y 46.8659, Z -8.0000, A 0.000, B 0.000, C 0.000 }
gfCNCPoint6[4250] = {X 95.6389, Y 47.6618, Z -8.0000, A 0.000, B 0.000, C 0.000 }
gfCNCPoint6[4251] = {X 94.9685, Y 48.3258, Z -8.0000, A 0.000, B 0.000, C 0.000 }
gfCNCPoint6[4252] = {X 94.1677, Y 48.8251, Z -8.0000, A 0.000, B 0.000, C 0.000 }
gfCNCPoint6[4253] = {X 93.2764, Y 49.1350, Z -8.0000, A 0.000, B 0.000, C 0.000 }
gfCNCPoint6[4254] = {X 92.3385, Y 49.2400, Z -8.0000, A 0.000, B 0.000, C 0.000 }
gfCNCPoint6[4255] = {X 85.8951, Y 49.2400, Z -8.0000, A 0.000, B 0.000, C 0.000 }
gfCNCPoint6[4256] = {X 84.9564, Y 49.1348, Z -8.0000, A 0.000, B 0.000, C 0.000 }
gfCNCPoint6[4257] = {X 84.0643, Y 48.8244, Z -8.0000, A 0.000, B 0.000, C 0.000 }
gfCNCPoint6[4258] = {X 83.2631, Y 48.3242, Z -8.0000, A 0.000, B 0.000, C 0.000 }
gfCNCPoint6[4259] = {X 82.5924, Y 47.6590, Z -8.0000, A 0.000, B 0.000, C 0.000 }
gfCNCPoint6[4260] = {X 82.0857, Y 46.8618, Z -8.0000, A 0.000, B 0.000, C 0.000 }
gfCNCPoint6[4261] = {X 81.7681, Y 45.9723, Z -8.0000, A 0.000, B 0.000, C 0.000 }
gfCNCPoint6[4262] = {X 81.6552, Y 45.0345, Z -8.0000, A 0.000, B 0.000, C 0.000 }
gfCNCPoint6[4263] = {X 81.6551, Y 44.2077, Z -8.0000, A 0.000, B 0.000, C 0.000 }
gfCNCPoint6[4264] = {X 81.7596, Y 43.2862, Z -8.0000, A 0.000, B 0.000, C 0.000 }
gfCNCPoint6[4265] = {X 82.0597, Y 42.4087, Z -8.0000, A 0.000, B 0.000, C 0.000 }
gfCNCPoint6[4266] = {X 82.5411, Y 41.6161, Z -8.0000, A 0.000, B 0.000, C 0.000 }
gfCNCPoint6[4267] = {X 83.1816, Y 40.9455, Z -8.0000, A 0.000, B 0.000, C 0.000 }
gfCNCPoint6[4268] = {X 83.1816, Y 28.5909, Z -8.0000, A 0.000, B 0.000, C 0.000 }
gfCNCPoint6[4269] = {X 79.1816, Y 28.5909, Z -8.0000, A 0.000, B 0.000, C 0.000 }
gfCNCPoint6[4270] = {X 83.2616, Y 28.5909, Z -8.0000, A 0.000, B 0.000, C 0.000 }
gfCNCPoint6[4271] = {X 83.2617, Y 16.1984, Z -8.0000, A 0.000, B 0.000, C 0.000 }
gfCNCPoint6[4272] = {X 82.6244, Y 15.5487, Z -8.0000, A 0.000, B 0.000, C 0.000 }
gfCNCPoint6[4273] = {X 82.1437, Y 14.7760, Z -8.0000, A 0.000, B 0.000, C 0.000 }
gfCNCPoint6[4274] = {X 81.8425, Y 13.9172, Z -8.0000, A 0.000, B 0.000, C 0.000 }
gfCNCPoint6[4275] = {X 81.7352, Y 13.0135, Z -8.0000, A 0.000, B 0.000, C 0.000 }
gfCNCPoint6[4276] = {X 81.7351, Y 12.1868, Z -8.0000, A 0.000, B 0.000, C 0.000 }
gfCNCPoint6[4277] = {X 81.8394, Y 11.2611, Z -8.0000, A 0.000, B 0.000, C 0.000 }
gfCNCPoint6[4278] = {X 82.1470, Y 10.3819, Z -8.0000, A 0.000, B 0.000, C 0.000 }
gfCNCPoint6[4279] = {X 82.6427, Y 9.5931, Z -8.0000, A 0.000, B 0.000, C 0.000 }
gfCNCPoint6[4280] = {X 83.3014, Y 8.9344, Z -8.0000, A 0.000, B 0.000, C 0.000 }
gfCNCPoint6[4281] = {X 84.0901, Y 8.4388, Z -8.0000, A 0.000, B 0.000, C 0.000 }
gfCNCPoint6[4282] = {X 84.9694, Y 8.1311, Z -8.0000, A 0.000, B 0.000, C 0.000 }
gfCNCPoint6[4283] = {X 85.8951, Y 8.0268, Z -8.0000, A 0.000, B 0.000, C 0.000 }
gfCNCPoint6[4284] = {X 94.0497, Y 8.0268, Z -8.0000, A 0.000, B 0.000, C 0.000 }
gfCNCPoint6[4285] = {X 94.9754, Y 8.1311, Z -8.0000, A 0.000, B 0.000, C 0.000 }
gfCNCPoint6[4286] = {X 95.8546, Y 8.4388, Z -8.0000, A 0.000, B 0.000, C 0.000 }
gfCNCPoint6[4287] = {X 96.6434, Y 8.9344, Z -8.0000, A 0.000, B 0.000, C 0.000 }
gfCNCPoint6[4288] = {X 97.3021, Y 9.5931, Z -8.0000, A 0.000, B 0.000, C 0.000 }
gfCNCPoint6[4289] = {X 97.7977, Y 10.3819, Z -8.0000, A 0.000, B 0.000, C 0.000 }
gfCNCPoint6[4290] = {X 98.1054, Y 11.2611, Z -8.0000, A 0.000, B 0.000, C 0.000 }
gfCNCPoint6[4291] = {X 98.2097, Y 12.1868, Z -8.0000, A 0.000, B 0.000, C 0.000 }
gfCNCPoint6[4292] = {X 98.2097, Y 12.9782, Z -8.0000, A 0.000, B 0.000, C 0.000 }
gfCNCPoint6[4293] = {X 98.1344, Y 13.7656, Z -8.0000, A 0.000, B 0.000, C 0.000 }
gfCNCPoint6[4294] = {X 97.9115, Y 14.5245, Z -8.0000, A 0.000, B 0.000, C 0.000 }
gfCNCPoint6[4295] = {X 97.5490, Y 15.2275, Z -8.0000, A 0.000, B 0.000, C 0.000 }
gfCNCPoint6[4296] = {X 101.8774, Y 25.9521, Z -8.0000, A 0.000, B 0.000, C 0.000 }
gfCNCPoint6[4297] = {X 106.1946, Y 15.2051, Z -8.0000, A 0.000, B 0.000, C 0.000 }
gfCNCPoint6[4298] = {X 105.8446, Y 14.5199, Z -8.0000, A 0.000, B 0.000, C 0.000 }
gfCNCPoint6[4299] = {X 105.6267, Y 13.7819, Z -8.0000, A 0.000, B 0.000, C 0.000 }
gfCNCPoint6[4300] = {X 105.5485, Y 13.0164, Z -8.0000, A 0.000, B 0.000, C 0.000 }
gfCNCPoint6[4301] = {X 105.5483, Y 12.1868, Z -8.0000, A 0.000, B 0.000, C 0.000 }
gfCNCPoint6[4302] = {X 105.6526, Y 11.2611, Z -8.0000, A 0.000, B 0.000, C 0.000 }
gfCNCPoint6[4303] = {X 105.9602, Y 10.3819, Z -8.0000, A 0.000, B 0.000, C 0.000 }
gfCNCPoint6[4304] = {X 106.4559, Y 9.5931, Z -8.0000, A 0.000, B 0.000, C 0.000 }
gfCNCPoint6[4305] = {X 107.1146, Y 8.9344, Z -8.0000, A 0.000, B 0.000, C 0.000 }
gfCNCPoint6[4306] = {X 107.9033, Y 8.4388, Z -8.0000, A 0.000, B 0.000, C 0.000 }
gfCNCPoint6[4307] = {X 108.7826, Y 8.1311, Z -8.0000, A 0.000, B 0.000, C 0.000 }
gfCNCPoint6[4308] = {X 109.7083, Y 8.0268, Z -8.0000, A 0.000, B 0.000, C 0.000 }
gfCNCPoint6[4309] = {X 117.7916, Y 8.0268, Z -8.0000, A 0.000, B 0.000, C 0.000 }
gfCNCPoint6[4310] = {X 118.7173, Y 8.1311, Z -8.0000, A 0.000, B 0.000, C 0.000 }
gfCNCPoint6[4311] = {X 119.5965, Y 8.4388, Z -8.0000, A 0.000, B 0.000, C 0.000 }
gfCNCPoint6[4312] = {X 120.3853, Y 8.9344, Z -8.0000, A 0.000, B 0.000, C 0.000 }
gfCNCPoint6[4313] = {X 121.0440, Y 9.5931, Z -8.0000, A 0.000, B 0.000, C 0.000 }
gfCNCPoint6[4314] = {X 121.5396, Y 10.3819, Z -8.0000, A 0.000, B 0.000, C 0.000 }
gfCNCPoint6[4315] = {X 121.8473, Y 11.2611, Z -8.0000, A 0.000, B 0.000, C 0.000 }
gfCNCPoint6[4316] = {X 121.9516, Y 12.1868, Z -8.0000, A 0.000, B 0.000, C 0.000 }
gfCNCPoint6[4317] = {X 121.9516, Y 12.9782, Z -8.0000, A 0.000, B 0.000, C 0.000 }
gfCNCPoint6[4318] = {X 121.8501, Y 13.8913, Z -8.0000, A 0.000, B 0.000, C 0.000 }
gfCNCPoint6[4319] = {X 121.5506, Y 14.7599, Z -8.0000, A 0.000, B 0.000, C 0.000 }
gfCNCPoint6[4320] = {X 121.0678, Y 15.5416, Z -8.0000, A 0.000, B 0.000, C 0.000 }
gfCNCPoint6[4321] = {X 120.4251, Y 16.1983, Z -8.0000, A 0.000, B 0.000, C 0.000 }
gfCNCPoint6[4322] = {X 120.4253, Y 40.9901, Z -8.0000, A 0.000, B 0.000, C 0.000 }
gfCNCPoint6[4323] = {X 120.5195, Y 41.0681, Z -8.0000, A 0.000, B 0.000, C 0.000 }
gfCNCPoint6[4324] = {X 121.1189, Y 41.7119, Z -8.0000, A 0.000, B 0.000, C 0.000 }
gfCNCPoint6[4325] = {X 121.5696, Y 42.4674, Z -8.0000, A 0.000, B 0.000, C 0.000 }
gfCNCPoint6[4326] = {X 121.8513, Y 43.3007, Z -8.0000, A 0.000, B 0.000, C 0.000 }
gfCNCPoint6[4327] = {X 121.9514, Y 44.1747, Z -8.0000, A 0.000, B 0.000, C 0.000 }
gfCNCPoint6[4328] = {X 121.9516, Y 45.0000, Z -8.0000, A 0.000, B 0.000, C 0.000 }
gfCNCPoint6[4329] = {X 121.8473, Y 45.9257, Z -8.0000, A 0.000, B 0.000, C 0.000 }
gfCNCPoint6[4330] = {X 121.5396, Y 46.8050, Z -8.0000, A 0.000, B 0.000, C 0.000 }
gfCNCPoint6[4331] = {X 121.0440, Y 47.5937, Z -8.0000, A 0.000, B 0.000, C 0.000 }
gfCNCPoint6[4332] = {X 120.3853, Y 48.2524, Z -8.0000, A 0.000, B 0.000, C 0.000 }
gfCNCPoint6[4333] = {X 119.5965, Y 48.7480, Z -8.0000, A 0.000, B 0.000, C 0.000 }
gfCNCPoint6[4334] = {X 118.7173, Y 49.0557, Z -8.0000, A 0.000, B 0.000, C 0.000 }
gfCNCPoint6[4335] = {X 117.7916, Y 49.1600, Z -8.0000, A 0.000, B 0.000, C 0.000 }
gfCNCPoint6[4336] = {X 111.9185, Y 49.1600, Z -8.0000, A 0.000, B 0.000, C 0.000 }
gfCNCPoint6[4337] = {X 110.9974, Y 49.0567, Z -8.0000, A 0.000, B 0.000, C 0.000 }
gfCNCPoint6[4338] = {X 110.1220, Y 48.7521, Z -8.0000, A 0.000, B 0.000, C 0.000 }
gfCNCPoint6[4339] = {X 109.3358, Y 48.2612, Z -8.0000, A 0.000, B 0.000, C 0.000 }
gfCNCPoint6[4340] = {X 108.6778, Y 47.6084, Z -8.0000, A 0.000, B 0.000, C 0.000 }
gfCNCPoint6[4341] = {X 108.1807, Y 46.8261, Z -8.0000, A 0.000, B 0.000, C 0.000 }
gfCNCPoint6[4342] = {X 107.8691, Y 45.9531, Z -8.0000, A 0.000, B 0.000, C 0.000 }
gfCNCPoint6[4343] = {X 107.7586, Y 45.0328, Z -8.0000, A 0.000, B 0.000, C 0.000 }
gfCNCPoint6[4344] = {X 107.7585, Y 44.1753, Z -8.0000, A 0.000, B 0.000, C 0.000 }
gfCNCPoint6[4345] = {X 107.7922, Y 43.6578, Z -8.0000, A 0.000, B 0.000, C 0.000 }
gfCNCPoint6[4346] = {X 107.8928, Y 43.1491, Z -8.0000, A 0.000, B 0.000, C 0.000 }
gfCNCPoint6[4347] = {X 108.0555, Y 42.6651, Z -8.0000, A 0.000, B 0.000, C 0.000 }
gfCNCPoint6[4348] = {X 108.2787, Y 42.2059, Z -8.0000, A 0.000, B 0.000, C 0.000 }
gfCNCPoint6[4349] = {X 108.7357, Y 41.5320, Z -8.0000, A 0.000, B 0.000, C 0.000 }
gfCNCPoint6[4350] = {X 109.2846, Y 40.9305, Z -8.0000, A 0.000, B 0.000, C 0.000 }
gfCNCPoint6[4351] = {X 109.2845, Y 39.0829, Z -8.0000, A 0.000, B 0.000, C 0.000 }
gfCNCPoint6[4352] = {X 109.0402, Y 39.0829, Z -8.0000, A 0.000, B 0.000, C 0.000 }
gfCNCPoint6[4353] = {X 105.9641, Y 46.5999, Z -8.0000, A 0.000, B 0.000, C 0.000 }
gfCNCPoint6[4354] = {X 105.6077, Y 47.2737, Z -8.0000, A 0.000, B 0.000, C 0.000 }
gfCNCPoint6[4355] = {X 105.1344, Y 47.8711, Z -8.0000, A 0.000, B 0.000, C 0.000 }
gfCNCPoint6[4356] = {X 104.5601, Y 48.3721, Z -8.0000, A 0.000, B 0.000, C 0.000 }
gfCNCPoint6[4357] = {X 103.9040, Y 48.7600, Z -8.0000, A 0.000, B 0.000, C 0.000 }
gfCNCPoint6[4358] = {X 102.9952, Y 49.0678, Z -8.0000, A 0.000, B 0.000, C 0.000 }
gfCNCPoint6[4359] = {X 102.0400, Y 49.1592, Z -8.0000, A 0.000, B 0.000, C 0.000 }
gfCNCPoint6[4360] = {X 101.0894, Y 49.0293, Z -8.0000, A 0.000, B 0.000, C 0.000 }
gfCNCPoint6[4361] = {X 100.1937, Y 48.6850, Z -8.0000, A 0.000, B 0.000, C 0.000 }
gfCNCPoint6[4362] = {X 99.4008, Y 48.1448, Z -8.0000, A 0.000, B 0.000, C 0.000 }
gfCNCPoint6[4363] = {X 98.7527, Y 47.4372, Z -8.0000, A 0.000, B 0.000, C 0.000 }
gfCNCPoint6[4364] = {X 98.2840, Y 46.5999, Z -8.0000, A 0.000, B 0.000, C 0.000 }
gfCNCPoint6[4365] = {X 94.9723, Y 38.5008, Z -8.0000, A 0.000, B 0.000, C 0.000 }
gfCNCPoint6[4366] = {X 94.9724, Y 40.9786, Z -8.0000, A 0.000, B 0.000, C 0.000 }
gfCNCPoint6[4367] = {X 95.5098, Y 41.5146, Z -8.0000, A 0.000, B 0.000, C 0.000 }
gfCNCPoint6[4368] = {X 95.9430, Y 42.1378, Z -8.0000, A 0.000, B 0.000, C 0.000 }
gfCNCPoint6[4369] = {X 96.1834, Y 42.6316, Z -8.0000, A 0.000, B 0.000, C 0.000 }
gfCNCPoint6[4370] = {X 96.3578, Y 43.1523, Z -8.0000, A 0.000, B 0.000, C 0.000 }
gfCNCPoint6[4371] = {X 96.4615, Y 43.6756, Z -8.0000, A 0.000, B 0.000, C 0.000 }
gfCNCPoint6[4372] = {X 96.4985, Y 44.2078, Z -8.0000, A 0.000, B 0.000, C 0.000 }
gfCNCPoint6[4373] = {X 96.4983, Y 45.0400, Z -8.0000, A 0.000, B 0.000, C 0.000 }
gfCNCPoint6[4374] = {X 96.3865, Y 45.9591, Z -8.0000, A 0.000, B 0.000, C 0.000 }
gfCNCPoint6[4375] = {X 96.0741, Y 46.8306, Z -8.0000, A 0.000, B 0.000, C 0.000 }
gfCNCPoint6[4376] = {X 95.5767, Y 47.6115, Z -8.0000, A 0.000, B 0.000, C 0.000 }
gfCNCPoint6[4377] = {X 94.9188, Y 48.2631, Z -8.0000, A 0.000, B 0.000, C 0.000 }
gfCNCPoint6[4378] = {X 94.1332, Y 48.7530, Z -8.0000, A 0.000, B 0.000, C 0.000 }
gfCNCPoint6[4379] = {X 93.2587, Y 49.0570, Z -8.0000, A 0.000, B 0.000, C 0.000 }
gfCNCPoint6[4380] = {X 92.3385, Y 49.1600, Z -8.0000, A 0.000, B 0.000, C 0.000 }
gfCNCPoint6[4381] = {X 85.8951, Y 49.1600, Z -8.0000, A 0.000, B 0.000, C 0.000 }
gfCNCPoint6[4382] = {X 84.9741, Y 49.0568, Z -8.0000, A 0.000, B 0.000, C 0.000 }
gfCNCPoint6[4383] = {X 84.0988, Y 48.7522, Z -8.0000, A 0.000, B 0.000, C 0.000 }
gfCNCPoint6[4384] = {X 83.3127, Y 48.2614, Z -8.0000, A 0.000, B 0.000, C 0.000 }
gfCNCPoint6[4385] = {X 82.6547, Y 47.6088, Z -8.0000, A 0.000, B 0.000, C 0.000 }
gfCNCPoint6[4386] = {X 82.1576, Y 46.8267, Z -8.0000, A 0.000, B 0.000, C 0.000 }
gfCNCPoint6[4387] = {X 81.8459, Y 45.9539, Z -8.0000, A 0.000, B 0.000, C 0.000 }
gfCNCPoint6[4388] = {X 81.7352, Y 45.0338, Z -8.0000, A 0.000, B 0.000, C 0.000 }
gfCNCPoint6[4389] = {X 81.7351, Y 44.2081, Z -8.0000, A 0.000, B 0.000, C 0.000 }
gfCNCPoint6[4390] = {X 81.8397, Y 43.2947, Z -8.0000, A 0.000, B 0.000, C 0.000 }
gfCNCPoint6[4391] = {X 82.1400, Y 42.4259, Z -8.0000, A 0.000, B 0.000, C 0.000 }
gfCNCPoint6[4392] = {X 82.6216, Y 41.6428, Z -8.0000, A 0.000, B 0.000, C 0.000 }
gfCNCPoint6[4393] = {X 83.2616, Y 40.9829, Z -8.0000, A 0.000, B 0.000, C 0.000 }
gfCNCPoint6[4394] = {X 83.2616, Y 28.5909, Z -8.0000, A 0.000, B 0.000, C 0.000 }
gfCNCPoint6[4395] = {X 79.2616, Y 28.5909, Z -8.0000, A 0.000, B 0.000, C 0.000 }
gfCNCPoint6[4396] = {X 83.3416, Y 28.5909, Z -8.0000, A 0.000, B 0.000, C 0.000 }
gfCNCPoint6[4397] = {X 83.3417, Y 16.1602, Z -8.0000, A 0.000, B 0.000, C 0.000 }
gfCNCPoint6[4398] = {X 82.7049, Y 15.5215, Z -8.0000, A 0.000, B 0.000, C 0.000 }
gfCNCPoint6[4399] = {X 82.2240, Y 14.7584, Z -8.0000, A 0.000, B 0.000, C 0.000 }
gfCNCPoint6[4400] = {X 81.9226, Y 13.9083, Z -8.0000, A 0.000, B 0.000, C 0.000 }
gfCNCPoint6[4401] = {X 81.8152, Y 13.0128, Z -8.0000, A 0.000, B 0.000, C 0.000 }
gfCNCPoint6[4402] = {X 81.8151, Y 12.1868, Z -8.0000, A 0.000, B 0.000, C 0.000 }
gfCNCPoint6[4403] = {X 81.9174, Y 11.2789, Z -8.0000, A 0.000, B 0.000, C 0.000 }
gfCNCPoint6[4404] = {X 82.2191, Y 10.4166, Z -8.0000, A 0.000, B 0.000, C 0.000 }
gfCNCPoint6[4405] = {X 82.7052, Y 9.6430, Z -8.0000, A 0.000, B 0.000, C 0.000 }
gfCNCPoint6[4406] = {X 83.3512, Y 8.9969, Z -8.0000, A 0.000, B 0.000, C 0.000 }
gfCNCPoint6[4407] = {X 84.1248, Y 8.5109, Z -8.0000, A 0.000, B 0.000, C 0.000 }
gfCNCPoint6[4408] = {X 84.9872, Y 8.2091, Z -8.0000, A 0.000, B 0.000, C 0.000 }
gfCNCPoint6[4409] = {X 85.8951, Y 8.1068, Z -8.0000, A 0.000, B 0.000, C 0.000 }
gfCNCPoint6[4410] = {X 94.0497, Y 8.1068, Z -8.0000, A 0.000, B 0.000, C 0.000 }
gfCNCPoint6[4411] = {X 94.9576, Y 8.2091, Z -8.0000, A 0.000, B 0.000, C 0.000 }
gfCNCPoint6[4412] = {X 95.8199, Y 8.5109, Z -8.0000, A 0.000, B 0.000, C 0.000 }
gfCNCPoint6[4413] = {X 96.5935, Y 8.9969, Z -8.0000, A 0.000, B 0.000, C 0.000 }
gfCNCPoint6[4414] = {X 97.2395, Y 9.6430, Z -8.0000, A 0.000, B 0.000, C 0.000 }
gfCNCPoint6[4415] = {X 97.7256, Y 10.4166, Z -8.0000, A 0.000, B 0.000, C 0.000 }
gfCNCPoint6[4416] = {X 98.0274, Y 11.2789, Z -8.0000, A 0.000, B 0.000, C 0.000 }
gfCNCPoint6[4417] = {X 98.1297, Y 12.1868, Z -8.0000, A 0.000, B 0.000, C 0.000 }
gfCNCPoint6[4418] = {X 98.1297, Y 12.9782, Z -8.0000, A 0.000, B 0.000, C 0.000 }
gfCNCPoint6[4419] = {X 98.0632, Y 13.7115, Z -8.0000, A 0.000, B 0.000, C 0.000 }
gfCNCPoint6[4420] = {X 97.8660, Y 14.4210, Z -8.0000, A 0.000, B 0.000, C 0.000 }
gfCNCPoint6[4421] = {X 97.5444, Y 15.0835, Z -8.0000, A 0.000, B 0.000, C 0.000 }
gfCNCPoint6[4422] = {X 97.4978, Y 15.1590, Z -8.0000, A 0.000, B 0.000, C 0.000 }
gfCNCPoint6[4423] = {X 97.4496, Y 15.2334, Z -8.0000, A 0.000, B 0.000, C 0.000 }
gfCNCPoint6[4424] = {X 97.4867, Y 15.2811, Z -8.0000, A 0.000, B 0.000, C 0.000 }
gfCNCPoint6[4425] = {X 101.8776, Y 26.1664, Z -8.0000, A 0.000, B 0.000, C 0.000 }
gfCNCPoint6[4426] = {X 106.2843, Y 15.1967, Z -8.0000, A 0.000, B 0.000, C 0.000 }
gfCNCPoint6[4427] = {X 106.2407, Y 15.1280, Z -8.0000, A 0.000, B 0.000, C 0.000 }
gfCNCPoint6[4428] = {X 106.1985, Y 15.0584, Z -8.0000, A 0.000, B 0.000, C 0.000 }
gfCNCPoint6[4429] = {X 105.8895, Y 14.4145, Z -8.0000, A 0.000, B 0.000, C 0.000 }
gfCNCPoint6[4430] = {X 105.6975, Y 13.7265, Z -8.0000, A 0.000, B 0.000, C 0.000 }
gfCNCPoint6[4431] = {X 105.6285, Y 13.0157, Z -8.0000, A 0.000, B 0.000, C 0.000 }
gfCNCPoint6[4432] = {X 105.6283, Y 12.1868, Z -8.0000, A 0.000, B 0.000, C 0.000 }
gfCNCPoint6[4433] = {X 105.7306, Y 11.2789, Z -8.0000, A 0.000, B 0.000, C 0.000 }
gfCNCPoint6[4434] = {X 106.0323, Y 10.4166, Z -8.0000, A 0.000, B 0.000, C 0.000 }
gfCNCPoint6[4435] = {X 106.5184, Y 9.6430, Z -8.0000, A 0.000, B 0.000, C 0.000 }
gfCNCPoint6[4436] = {X 107.1644, Y 8.9969, Z -8.0000, A 0.000, B 0.000, C 0.000 }
gfCNCPoint6[4437] = {X 107.9380, Y 8.5109, Z -8.0000, A 0.000, B 0.000, C 0.000 }
gfCNCPoint6[4438] = {X 108.8004, Y 8.2091, Z -8.0000, A 0.000, B 0.000, C 0.000 }
gfCNCPoint6[4439] = {X 109.7083, Y 8.1068, Z -8.0000, A 0.000, B 0.000, C 0.000 }
gfCNCPoint6[4440] = {X 117.7916, Y 8.1068, Z -8.0000, A 0.000, B 0.000, C 0.000 }
gfCNCPoint6[4441] = {X 118.6995, Y 8.2091, Z -8.0000, A 0.000, B 0.000, C 0.000 }
gfCNCPoint6[4442] = {X 119.5618, Y 8.5109, Z -8.0000, A 0.000, B 0.000, C 0.000 }
gfCNCPoint6[4443] = {X 120.3354, Y 8.9969, Z -8.0000, A 0.000, B 0.000, C 0.000 }
gfCNCPoint6[4444] = {X 120.9814, Y 9.6430, Z -8.0000, A 0.000, B 0.000, C 0.000 }
gfCNCPoint6[4445] = {X 121.4675, Y 10.4166, Z -8.0000, A 0.000, B 0.000, C 0.000 }
gfCNCPoint6[4446] = {X 121.7693, Y 11.2789, Z -8.0000, A 0.000, B 0.000, C 0.000 }
gfCNCPoint6[4447] = {X 121.8716, Y 12.1868, Z -8.0000, A 0.000, B 0.000, C 0.000 }
gfCNCPoint6[4448] = {X 121.8716, Y 12.9782, Z -8.0000, A 0.000, B 0.000, C 0.000 }
gfCNCPoint6[4449] = {X 121.7699, Y 13.8830, Z -8.0000, A 0.000, B 0.000, C 0.000 }
gfCNCPoint6[4450] = {X 121.4702, Y 14.7427, Z -8.0000, A 0.000, B 0.000, C 0.000 }
gfCNCPoint6[4451] = {X 120.9872, Y 15.5146, Z -8.0000, A 0.000, B 0.000, C 0.000 }
gfCNCPoint6[4452] = {X 120.3451, Y 16.1601, Z -8.0000, A 0.000, B 0.000, C 0.000 }
gfCNCPoint6[4453] = {X 120.3453, Y 41.0277, Z -8.0000, A 0.000, B 0.000, C 0.000 }
gfCNCPoint6[4454] = {X 120.4678, Y 41.1291, Z -8.0000, A 0.000, B 0.000, C 0.000 }
gfCNCPoint6[4455] = {X 121.0554, Y 41.7605, Z -8.0000, A 0.000, B 0.000, C 0.000 }
gfCNCPoint6[4456] = {X 121.4971, Y 42.5013, Z -8.0000, A 0.000, B 0.000, C 0.000 }
gfCNCPoint6[4457] = {X 121.7732, Y 43.3184, Z -8.0000, A 0.000, B 0.000, C 0.000 }
gfCNCPoint6[4458] = {X 121.8714, Y 44.1754, Z -8.0000, A 0.000, B 0.000, C 0.000 }
gfCNCPoint6[4459] = {X 121.8716, Y 45.0000, Z -8.0000, A 0.000, B 0.000, C 0.000 }
gfCNCPoint6[4460] = {X 121.7693, Y 45.9079, Z -8.0000, A 0.000, B 0.000, C 0.000 }
gfCNCPoint6[4461] = {X 121.4675, Y 46.7702, Z -8.0000, A 0.000, B 0.000, C 0.000 }
gfCNCPoint6[4462] = {X 120.9814, Y 47.5438, Z -8.0000, A 0.000, B 0.000, C 0.000 }
gfCNCPoint6[4463] = {X 120.3354, Y 48.1899, Z -8.0000, A 0.000, B 0.000, C 0.000 }
gfCNCPoint6[4464] = {X 119.5618, Y 48.6760, Z -8.0000, A 0.000, B 0.000, C 0.000 }
gfCNCPoint6[4465] = {X 118.6995, Y 48.9777, Z -8.0000, A 0.000, B 0.000, C 0.000 }
gfCNCPoint6[4466] = {X 117.7916, Y 49.0800, Z -8.0000, A 0.000, B 0.000, C 0.000 }
gfCNCPoint6[4467] = {X 111.9185, Y 49.0800, Z -8.0000, A 0.000, B 0.000, C 0.000 }
gfCNCPoint6[4468] = {X 111.0151, Y 48.9787, Z -8.0000, A 0.000, B 0.000, C 0.000 }
gfCNCPoint6[4469] = {X 110.1565, Y 48.6799, Z -8.0000, A 0.000, B 0.000, C 0.000 }
gfCNCPoint6[4470] = {X 109.3855, Y 48.1985, Z -8.0000, A 0.000, B 0.000, C 0.000 }
gfCNCPoint6[4471] = {X 108.7401, Y 47.5582, Z -8.0000, A 0.000, B 0.000, C 0.000 }
gfCNCPoint6[4472] = {X 108.2526, Y 46.7909, Z -8.0000, A 0.000, B 0.000, C 0.000 }
gfCNCPoint6[4473] = {X 107.9470, Y 45.9348, Z -8.0000, A 0.000, B 0.000, C 0.000 }
gfCNCPoint6[4474] = {X 107.8386, Y 45.0322, Z -8.0000, A 0.000, B 0.000, C 0.000 }
gfCNCPoint6[4475] = {X 107.8385, Y 44.1753, Z -8.0000, A 0.000, B 0.000, C 0.000 }
gfCNCPoint6[4476] = {X 107.8715, Y 43.6682, Z -8.0000, A 0.000, B 0.000, C 0.000 }
gfCNCPoint6[4477] = {X 107.9701, Y 43.1697, Z -8.0000, A 0.000, B 0.000, C 0.000 }
gfCNCPoint6[4478] = {X 108.1295, Y 42.6954, Z -8.0000, A 0.000, B 0.000, C 0.000 }
gfCNCPoint6[4479] = {X 108.3483, Y 42.2454, Z -8.0000, A 0.000, B 0.000, C 0.000 }
gfCNCPoint6[4480] = {X 108.8093, Y 41.5678, Z -8.0000, A 0.000, B 0.000, C 0.000 }
gfCNCPoint6[4481] = {X 109.3646, Y 40.9650, Z -8.0000, A 0.000, B 0.000, C 0.000 }
gfCNCPoint6[4482] = {X 109.3645, Y 39.0029, Z -8.0000, A 0.000, B 0.000, C 0.000 }
gfCNCPoint6[4483] = {X 108.9865, Y 39.0029, Z -8.0000, A 0.000, B 0.000, C 0.000 }
gfCNCPoint6[4484] = {X 105.8902, Y 46.5692, Z -8.0000, A 0.000, B 0.000, C 0.000 }
gfCNCPoint6[4485] = {X 105.5407, Y 47.2300, Z -8.0000, A 0.000, B 0.000, C 0.000 }
gfCNCPoint6[4486] = {X 105.0765, Y 47.8159, Z -8.0000, A 0.000, B 0.000, C 0.000 }
gfCNCPoint6[4487] = {X 104.5133, Y 48.3073, Z -8.0000, A 0.000, B 0.000, C 0.000 }
gfCNCPoint6[4488] = {X 103.8698, Y 48.6877, Z -8.0000, A 0.000, B 0.000, C 0.000 }
gfCNCPoint6[4489] = {X 102.9784, Y 48.9895, Z -8.0000, A 0.000, B 0.000, C 0.000 }
gfCNCPoint6[4490] = {X 102.0417, Y 49.0792, Z -8.0000, A 0.000, B 0.000, C 0.000 }
gfCNCPoint6[4491] = {X 101.1093, Y 48.9518, Z -8.0000, A 0.000, B 0.000, C 0.000 }
gfCNCPoint6[4492] = {X 100.2309, Y 48.6142, Z -8.0000, A 0.000, B 0.000, C 0.000 }
gfCNCPoint6[4493] = {X 99.4532, Y 48.0843, Z -8.0000, A 0.000, B 0.000, C 0.000 }
gfCNCPoint6[4494] = {X 98.8176, Y 47.3903, Z -8.0000, A 0.000, B 0.000, C 0.000 }
gfCNCPoint6[4495] = {X 98.3579, Y 46.5692, Z -8.0000, A 0.000, B 0.000, C 0.000 }
gfCNCPoint6[4496] = {X 94.8932, Y 38.0959, Z -8.0000, A 0.000, B 0.000, C 0.000 }
gfCNCPoint6[4497] = {X 94.8923, Y 38.2309, Z -8.0000, A 0.000, B 0.000, C 0.000 }
gfCNCPoint6[4498] = {X 94.8924, Y 41.0163, Z -8.0000, A 0.000, B 0.000, C 0.000 }
gfCNCPoint6[4499] = {X 95.4364, Y 41.5516, Z -8.0000, A 0.000, B 0.000, C 0.000 }
gfCNCPoint6[4500] = {X 95.8735, Y 42.1774, Z -8.0000, A 0.000, B 0.000, C 0.000 }
gfCNCPoint6[4501] = {X 96.1093, Y 42.6618, Z -8.0000, A 0.000, B 0.000, C 0.000 }
gfCNCPoint6[4502] = {X 96.2805, Y 43.1727, Z -8.0000, A 0.000, B 0.000, C 0.000 }
gfCNCPoint6[4503] = {X 96.3822, Y 43.6862, Z -8.0000, A 0.000, B 0.000, C 0.000 }
gfCNCPoint6[4504] = {X 96.4185, Y 44.2083, Z -8.0000, A 0.000, B 0.000, C 0.000 }
gfCNCPoint6[4505] = {X 96.4184, Y 45.0392, Z -8.0000, A 0.000, B 0.000, C 0.000 }
gfCNCPoint6[4506] = {X 96.3086, Y 45.9406, Z -8.0000, A 0.000, B 0.000, C 0.000 }
gfCNCPoint6[4507] = {X 96.0023, Y 46.7954, Z -8.0000, A 0.000, B 0.000, C 0.000 }
gfCNCPoint6[4508] = {X 95.5144, Y 47.5613, Z -8.0000, A 0.000, B 0.000, C 0.000 }
gfCNCPoint6[4509] = {X 94.8692, Y 48.2003, Z -8.0000, A 0.000, B 0.000, C 0.000 }
gfCNCPoint6[4510] = {X 94.0987, Y 48.6808, Z -8.0000, A 0.000, B 0.000, C 0.000 }
gfCNCPoint6[4511] = {X 93.2410, Y 48.9789, Z -8.0000, A 0.000, B 0.000, C 0.000 }
gfCNCPoint6[4512] = {X 92.3385, Y 49.0800, Z -8.0000, A 0.000, B 0.000, C 0.000 }
gfCNCPoint6[4513] = {X 85.8951, Y 49.0800, Z -8.0000, A 0.000, B 0.000, C 0.000 }
gfCNCPoint6[4514] = {X 84.9918, Y 48.9788, Z -8.0000, A 0.000, B 0.000, C 0.000 }
gfCNCPoint6[4515] = {X 84.1334, Y 48.6801, Z -8.0000, A 0.000, B 0.000, C 0.000 }
gfCNCPoint6[4516] = {X 83.3624, Y 48.1987, Z -8.0000, A 0.000, B 0.000, C 0.000 }
gfCNCPoint6[4517] = {X 82.7171, Y 47.5586, Z -8.0000, A 0.000, B 0.000, C 0.000 }
gfCNCPoint6[4518] = {X 82.2295, Y 46.7916, Z -8.0000, A 0.000, B 0.000, C 0.000 }
gfCNCPoint6[4519] = {X 81.9238, Y 45.9356, Z -8.0000, A 0.000, B 0.000, C 0.000 }
gfCNCPoint6[4520] = {X 81.8152, Y 45.0332, Z -8.0000, A 0.000, B 0.000, C 0.000 }
gfCNCPoint6[4521] = {X 81.8151, Y 44.2084, Z -8.0000, A 0.000, B 0.000, C 0.000 }
gfCNCPoint6[4522] = {X 81.9198, Y 43.3033, Z -8.0000, A 0.000, B 0.000, C 0.000 }
gfCNCPoint6[4523] = {X 82.2204, Y 42.4432, Z -8.0000, A 0.000, B 0.000, C 0.000 }
gfCNCPoint6[4524] = {X 82.7021, Y 41.6698, Z -8.0000, A 0.000, B 0.000, C 0.000 }
gfCNCPoint6[4525] = {X 83.3416, Y 41.0207, Z -8.0000, A 0.000, B 0.000, C 0.000 }
gfCNCPoint6[4526] = {X 83.3416, Y 28.5909, Z -8.0000, A 0.000, B 0.000, C 0.000 }
gfCNCPoint6[4527] = {X 79.3416, Y 28.5909, Z -8.0000, A 0.000, B 0.000, C 0.000 }
gfCNCPoint6[4528] = {X 83.4216, Y 28.5909, Z -8.0000, A 0.000, B 0.000, C 0.000 }
gfCNCPoint6[4529] = {X 83.4217, Y 16.1216, Z -8.0000, A 0.000, B 0.000, C 0.000 }
gfCNCPoint6[4530] = {X 82.7800, Y 15.4873, Z -8.0000, A 0.000, B 0.000, C 0.000 }
gfCNCPoint6[4531] = {X 82.2969, Y 14.7253, Z -8.0000, A 0.000, B 0.000, C 0.000 }
gfCNCPoint6[4532] = {X 81.9968, Y 13.8745, Z -8.0000, A 0.000, B 0.000, C 0.000 }
gfCNCPoint6[4533] = {X 81.8951, Y 12.9780, Z -8.0000, A 0.000, B 0.000, C 0.000 }
gfCNCPoint6[4534] = {X 81.8951, Y 12.1868, Z -8.0000, A 0.000, B 0.000, C 0.000 }
gfCNCPoint6[4535] = {X 81.9954, Y 11.2967, Z -8.0000, A 0.000, B 0.000, C 0.000 }
gfCNCPoint6[4536] = {X 82.2912, Y 10.4513, Z -8.0000, A 0.000, B 0.000, C 0.000 }
gfCNCPoint6[4537] = {X 82.7677, Y 9.6929, Z -8.0000, A 0.000, B 0.000, C 0.000 }
gfCNCPoint6[4538] = {X 83.4011, Y 9.0595, Z -8.0000, A 0.000, B 0.000, C 0.000 }
gfCNCPoint6[4539] = {X 84.1595, Y 8.5829, Z -8.0000, A 0.000, B 0.000, C 0.000 }
gfCNCPoint6[4540] = {X 85.0050, Y 8.2871, Z -8.0000, A 0.000, B 0.000, C 0.000 }
gfCNCPoint6[4541] = {X 85.8951, Y 8.1868, Z -8.0000, A 0.000, B 0.000, C 0.000 }
gfCNCPoint6[4542] = {X 94.0497, Y 8.1868, Z -8.0000, A 0.000, B 0.000, C 0.000 }
gfCNCPoint6[4543] = {X 94.9398, Y 8.2871, Z -8.0000, A 0.000, B 0.000, C 0.000 }
gfCNCPoint6[4544] = {X 95.7852, Y 8.5829, Z -8.0000, A 0.000, B 0.000, C 0.000 }
gfCNCPoint6[4545] = {X 96.5436, Y 9.0595, Z -8.0000, A 0.000, B 0.000, C 0.000 }
gfCNCPoint6[4546] = {X 97.1770, Y 9.6929, Z -8.0000, A 0.000, B 0.000, C 0.000 }
gfCNCPoint6[4547] = {X 97.6535, Y 10.4513, Z -8.0000, A 0.000, B 0.000, C 0.000 }
gfCNCPoint6[4548] = {X 97.9494, Y 11.2967, Z -8.0000, A 0.000, B 0.000, C 0.000 }
gfCNCPoint6[4549] = {X 98.0497, Y 12.1868, Z -8.0000, A 0.000, B 0.000, C 0.000 }
gfCNCPoint6[4550] = {X 98.0495, Y 13.0192, Z -8.0000, A 0.000, B 0.000, C 0.000 }
gfCNCPoint6[4551] = {X 97.9795, Y 13.7240, Z -8.0000, A 0.000, B 0.000, C 0.000 }
gfCNCPoint6[4552] = {X 97.7863, Y 14.4055, Z -8.0000, A 0.000, B 0.000, C 0.000 }
gfCNCPoint6[4553] = {X 97.4759, Y 15.0422, Z -8.0000, A 0.000, B 0.000, C 0.000 }
gfCNCPoint6[4554] = {X 97.4132, Y 15.1428, Z -8.0000, A 0.000, B 0.000, C 0.000 }
gfCNCPoint6[4555] = {X 97.3476, Y 15.2415, Z -8.0000, A 0.000, B 0.000, C 0.000 }
gfCNCPoint6[4556] = {X 97.4125, Y 15.3109, Z -8.0000, A 0.000, B 0.000, C 0.000 }
gfCNCPoint6[4557] = {X 98.2761, Y 17.4611, Z -8.0000, A 0.000, B 0.000, C 0.000 }
gfCNCPoint6[4558] = {X 101.8768, Y 26.3781, Z -8.0000, A 0.000, B 0.000, C 0.000 }
gfCNCPoint6[4559] = {X 101.9496, Y 26.2017, Z -8.0000, A 0.000, B 0.000, C 0.000 }
gfCNCPoint6[4560] = {X 105.7340, Y 16.7687, Z -8.0000, A 0.000, B 0.000, C 0.000 }
gfCNCPoint6[4561] = {X 106.3406, Y 15.2554, Z -8.0000, A 0.000, B 0.000, C 0.000 }
gfCNCPoint6[4562] = {X 106.3813, Y 15.1986, Z -8.0000, A 0.000, B 0.000, C 0.000 }
gfCNCPoint6[4563] = {X 106.3231, Y 15.1089, Z -8.0000, A 0.000, B 0.000, C 0.000 }
gfCNCPoint6[4564] = {X 106.2673, Y 15.0176, Z -8.0000, A 0.000, B 0.000, C 0.000 }
gfCNCPoint6[4565] = {X 105.9601, Y 14.3748, Z -8.0000, A 0.000, B 0.000, C 0.000 }
gfCNCPoint6[4566] = {X 105.7717, Y 13.6876, Z -8.0000, A 0.000, B 0.000, C 0.000 }
gfCNCPoint6[4567] = {X 105.7083, Y 12.9780, Z -8.0000, A 0.000, B 0.000, C 0.000 }
gfCNCPoint6[4568] = {X 105.7083, Y 12.1868, Z -8.0000, A 0.000, B 0.000, C 0.000 }
gfCNCPoint6[4569] = {X 105.8086, Y 11.2967, Z -8.0000, A 0.000, B 0.000, C 0.000 }
gfCNCPoint6[4570] = {X 106.1044, Y 10.4513, Z -8.0000, A 0.000, B 0.000, C 0.000 }
gfCNCPoint6[4571] = {X 106.5810, Y 9.6929, Z -8.0000, A 0.000, B 0.000, C 0.000 }
gfCNCPoint6[4572] = {X 107.2143, Y 9.0595, Z -8.0000, A 0.000, B 0.000, C 0.000 }
gfCNCPoint6[4573] = {X 107.9727, Y 8.5829, Z -8.0000, A 0.000, B 0.000, C 0.000 }
gfCNCPoint6[4574] = {X 108.8182, Y 8.2871, Z -8.0000, A 0.000, B 0.000, C 0.000 }
gfCNCPoint6[4575] = {X 109.7083, Y 8.1868, Z -8.0000, A 0.000, B 0.000, C 0.000 }
gfCNCPoint6[4576] = {X 117.7916, Y 8.1868, Z -8.0000, A 0.000, B 0.000, C 0.000 }
gfCNCPoint6[4577] = {X 118.6817, Y 8.2871, Z -8.0000, A 0.000, B 0.000, C 0.000 }
gfCNCPoint6[4578] = {X 119.5271, Y 8.5829, Z -8.0000, A 0.000, B 0.000, C 0.000 }
gfCNCPoint6[4579] = {X 120.2855, Y 9.0595, Z -8.0000, A 0.000, B 0.000, C 0.000 }
gfCNCPoint6[4580] = {X 120.9189, Y 9.6929, Z -8.0000, A 0.000, B 0.000, C 0.000 }
gfCNCPoint6[4581] = {X 121.3955, Y 10.4513, Z -8.0000, A 0.000, B 0.000, C 0.000 }
gfCNCPoint6[4582] = {X 121.6913, Y 11.2967, Z -8.0000, A 0.000, B 0.000, C 0.000 }
gfCNCPoint6[4583] = {X 121.7916, Y 12.1868, Z -8.0000, A 0.000, B 0.000, C 0.000 }
gfCNCPoint6[4584] = {X 121.7914, Y 13.0192, Z -8.0000, A 0.000, B 0.000, C 0.000 }
gfCNCPoint6[4585] = {X 121.6828, Y 13.9045, Z -8.0000, A 0.000, B 0.000, C 0.000 }
gfCNCPoint6[4586] = {X 121.3807, Y 14.7438, Z -8.0000, A 0.000, B 0.000, C 0.000 }
gfCNCPoint6[4587] = {X 120.9002, Y 15.4952, Z -8.0000, A 0.000, B 0.000, C 0.000 }
gfCNCPoint6[4588] = {X 120.2651, Y 16.1215, Z -8.0000, A 0.000, B 0.000, C 0.000 }
gfCNCPoint6[4589] = {X 120.2653, Y 41.0653, Z -8.0000, A 0.000, B 0.000, C 0.000 }
gfCNCPoint6[4590] = {X 120.4160, Y 41.1901, Z -8.0000, A 0.000, B 0.000, C 0.000 }
gfCNCPoint6[4591] = {X 120.9967, Y 41.8157, Z -8.0000, A 0.000, B 0.000, C 0.000 }
gfCNCPoint6[4592] = {X 121.4315, Y 42.5502, Z -8.0000, A 0.000, B 0.000, C 0.000 }
gfCNCPoint6[4593] = {X 121.7005, Y 43.3602, Z -8.0000, A 0.000, B 0.000, C 0.000 }
gfCNCPoint6[4594] = {X 121.7916, Y 44.2089, Z -8.0000, A 0.000, B 0.000, C 0.000 }
gfCNCPoint6[4595] = {X 121.7916, Y 45.0000, Z -8.0000, A 0.000, B 0.000, C 0.000 }
gfCNCPoint6[4596] = {X 121.6913, Y 45.8901, Z -8.0000, A 0.000, B 0.000, C 0.000 }
gfCNCPoint6[4597] = {X 121.3955, Y 46.7355, Z -8.0000, A 0.000, B 0.000, C 0.000 }
gfCNCPoint6[4598] = {X 120.9189, Y 47.4940, Z -8.0000, A 0.000, B 0.000, C 0.000 }
gfCNCPoint6[4599] = {X 120.2855, Y 48.1273, Z -8.0000, A 0.000, B 0.000, C 0.000 }
gfCNCPoint6[4600] = {X 119.5271, Y 48.6039, Z -8.0000, A 0.000, B 0.000, C 0.000 }
gfCNCPoint6[4601] = {X 118.6817, Y 48.8997, Z -8.0000, A 0.000, B 0.000, C 0.000 }
gfCNCPoint6[4602] = {X 117.7916, Y 49.0000, Z -8.0000, A 0.000, B 0.000, C 0.000 }
gfCNCPoint6[4603] = {X 111.9185, Y 49.0000, Z -8.0000, A 0.000, B 0.000, C 0.000 }
gfCNCPoint6[4604] = {X 111.0284, Y 48.8997, Z -8.0000, A 0.000, B 0.000, C 0.000 }
gfCNCPoint6[4605] = {X 110.1829, Y 48.6039, Z -8.0000, A 0.000, B 0.000, C 0.000 }
gfCNCPoint6[4606] = {X 109.4245, Y 48.1273, Z -8.0000, A 0.000, B 0.000, C 0.000 }
gfCNCPoint6[4607] = {X 108.7911, Y 47.4939, Z -8.0000, A 0.000, B 0.000, C 0.000 }
gfCNCPoint6[4608] = {X 108.3146, Y 46.7355, Z -8.0000, A 0.000, B 0.000, C 0.000 }
gfCNCPoint6[4609] = {X 108.0188, Y 45.8901, Z -8.0000, A 0.000, B 0.000, C 0.000 }
gfCNCPoint6[4610] = {X 107.9185, Y 45.0000, Z -8.0000, A 0.000, B 0.000, C 0.000 }
gfCNCPoint6[4611] = {X 107.9185, Y 44.1753, Z -8.0000, A 0.000, B 0.000, C 0.000 }
gfCNCPoint6[4612] = {X 107.9508, Y 43.6786, Z -8.0000, A 0.000, B 0.000, C 0.000 }
gfCNCPoint6[4613] = {X 108.0474, Y 43.1903, Z -8.0000, A 0.000, B 0.000, C 0.000 }
gfCNCPoint6[4614] = {X 108.2036, Y 42.7257, Z -8.0000, A 0.000, B 0.000, C 0.000 }
gfCNCPoint6[4615] = {X 108.4179, Y 42.2850, Z -8.0000, A 0.000, B 0.000, C 0.000 }
gfCNCPoint6[4616] = {X 108.4421, Y 42.2429, Z -8.0000, A 0.000, B 0.000, C 0.000 }
gfCNCPoint6[4617] = {X 108.4669, Y 42.2011, Z -8.0000, A 0.000, B 0.000, C 0.000 }
gfCNCPoint6[4618] = {X 108.9133, Y 41.5659, Z -8.0000, A 0.000, B 0.000, C 0.000 }
gfCNCPoint6[4619] = {X 109.4446, Y 40.9999, Z -8.0000, A 0.000, B 0.000, C 0.000 }
gfCNCPoint6[4620] = {X 109.4445, Y 38.9229, Z -8.0000, A 0.000, B 0.000, C 0.000 }
gfCNCPoint6[4621] = {X 108.9328, Y 38.9229, Z -8.0000, A 0.000, B 0.000, C 0.000 }
gfCNCPoint6[4622] = {X 105.8164, Y 46.5384, Z -8.0000, A 0.000, B 0.000, C 0.000 }
gfCNCPoint6[4623] = {X 105.3339, Y 47.3869, Z -8.0000, A 0.000, B 0.000, C 0.000 }
gfCNCPoint6[4624] = {X 104.6602, Y 48.0932, Z -8.0000, A 0.000, B 0.000, C 0.000 }
gfCNCPoint6[4625] = {X 103.8355, Y 48.6154, Z -8.0000, A 0.000, B 0.000, C 0.000 }
gfCNCPoint6[4626] = {X 102.9580, Y 48.9121, Z -8.0000, A 0.000, B 0.000, C 0.000 }
gfCNCPoint6[4627] = {X 102.0357, Y 48.9990, Z -8.0000, A 0.000, B 0.000, C 0.000 }
gfCNCPoint6[4628] = {X 101.1182, Y 48.8715, Z -8.0000, A 0.000, B 0.000, C 0.000 }
gfCNCPoint6[4629] = {X 100.2546, Y 48.5362, Z -8.0000, A 0.000, B 0.000, C 0.000 }
gfCNCPoint6[4630] = {X 99.4912, Y 48.0114, Z -8.0000, A 0.000, B 0.000, C 0.000 }
gfCNCPoint6[4631] = {X 98.8691, Y 47.3250, Z -8.0000, A 0.000, B 0.000, C 0.000 }
gfCNCPoint6[4632] = {X 98.4216, Y 46.5139, Z -8.0000, A 0.000, B 0.000, C 0.000 }
gfCNCPoint6[4633] = {X 94.8157, Y 37.6951, Z -8.0000, A 0.000, B 0.000, C 0.000 }
gfCNCPoint6[4634] = {X 94.8123, Y 38.2306, Z -8.0000, A 0.000, B 0.000, C 0.000 }
gfCNCPoint6[4635] = {X 94.8124, Y 41.0545, Z -8.0000, A 0.000, B 0.000, C 0.000 }
gfCNCPoint6[4636] = {X 95.3631, Y 41.5889, Z -8.0000, A 0.000, B 0.000, C 0.000 }
gfCNCPoint6[4637] = {X 95.8040, Y 42.2170, Z -8.0000, A 0.000, B 0.000, C 0.000 }
gfCNCPoint6[4638] = {X 96.0353, Y 42.6921, Z -8.0000, A 0.000, B 0.000, C 0.000 }
gfCNCPoint6[4639] = {X 96.2032, Y 43.1932, Z -8.0000, A 0.000, B 0.000, C 0.000 }
gfCNCPoint6[4640] = {X 96.3029, Y 43.6967, Z -8.0000, A 0.000, B 0.000, C 0.000 }
gfCNCPoint6[4641] = {X 96.3385, Y 44.2088, Z -8.0000, A 0.000, B 0.000, C 0.000 }
gfCNCPoint6[4642] = {X 96.3384, Y 45.0384, Z -8.0000, A 0.000, B 0.000, C 0.000 }
gfCNCPoint6[4643] = {X 96.2308, Y 45.9222, Z -8.0000, A 0.000, B 0.000, C 0.000 }
gfCNCPoint6[4644] = {X 95.9304, Y 46.7602, Z -8.0000, A 0.000, B 0.000, C 0.000 }
gfCNCPoint6[4645] = {X 95.4521, Y 47.5111, Z -8.0000, A 0.000, B 0.000, C 0.000 }
gfCNCPoint6[4646] = {X 94.8196, Y 48.1376, Z -8.0000, A 0.000, B 0.000, C 0.000 }
gfCNCPoint6[4647] = {X 94.0642, Y 48.6086, Z -8.0000, A 0.000, B 0.000, C 0.000 }
gfCNCPoint6[4648] = {X 93.2233, Y 48.9009, Z -8.0000, A 0.000, B 0.000, C 0.000 }
gfCNCPoint6[4649] = {X 92.3385, Y 49.0000, Z -8.0000, A 0.000, B 0.000, C 0.000 }
gfCNCPoint6[4650] = {X 85.8951, Y 49.0000, Z -8.0000, A 0.000, B 0.000, C 0.000 }
gfCNCPoint6[4651] = {X 85.0050, Y 48.8997, Z -8.0000, A 0.000, B 0.000, C 0.000 }
gfCNCPoint6[4652] = {X 84.1595, Y 48.6039, Z -8.0000, A 0.000, B 0.000, C 0.000 }
gfCNCPoint6[4653] = {X 83.4011, Y 48.1273, Z -8.0000, A 0.000, B 0.000, C 0.000 }
gfCNCPoint6[4654] = {X 82.7677, Y 47.4939, Z -8.0000, A 0.000, B 0.000, C 0.000 }
gfCNCPoint6[4655] = {X 82.2912, Y 46.7355, Z -8.0000, A 0.000, B 0.000, C 0.000 }
gfCNCPoint6[4656] = {X 81.9954, Y 45.8901, Z -8.0000, A 0.000, B 0.000, C 0.000 }
gfCNCPoint6[4657] = {X 81.8951, Y 45.0000, Z -8.0000, A 0.000, B 0.000, C 0.000 }
gfCNCPoint6[4658] = {X 81.8951, Y 44.2088, Z -8.0000, A 0.000, B 0.000, C 0.000 }
gfCNCPoint6[4659] = {X 81.9999, Y 43.3120, Z -8.0000, A 0.000, B 0.000, C 0.000 }
gfCNCPoint6[4660] = {X 82.3008, Y 42.4606, Z -8.0000, A 0.000, B 0.000, C 0.000 }
gfCNCPoint6[4661] = {X 82.7826, Y 41.6970, Z -8.0000, A 0.000, B 0.000, C 0.000 }
gfCNCPoint6[4662] = {X 83.4216, Y 41.0590, Z -8.0000, A 0.000, B 0.000, C 0.000 }
gfCNCPoint6[4663] = {X 83.4216, Y 28.5909, Z -8.0000, A 0.000, B 0.000, C 0.000 }
gfCNCPoint6[4664] = {X 79.3416, Y 28.5909, Z -8.0000, A 0.000, B 0.000, C 0.000 }
gfCNCPoint6[4665] = {X 79.3416, Y 28.5909, Z -5.0000, A 0.000, B 0.000, C 0.000 }
gfCNCPoint6[4666] = {X 79.3416, Y 28.5909, Z 11.0000, A 0.000, B 0.000, C 0.000 }
gfCNCPoint6[4667] = {X 136.1636, Y 30.3971, Z 11.0000, A 0.000, B 0.000, C 0.000 }
gfCNCPoint6[4668] = {X 136.1636, Y 30.3971, Z -5.0000, A 0.000, B 0.000, C 0.000 }
gfCNCPoint6[4669] = {X 136.1636, Y 30.3971, Z -8.0000, A 0.000, B 0.000, C 0.000 }
gfCNCPoint6[4670] = {X 140.2436, Y 30.3971, Z -8.0000, A 0.000, B 0.000, C 0.000 }
gfCNCPoint6[4671] = {X 140.2436, Y 19.8785, Z -8.0000, A 0.000, B 0.000, C 0.000 }
gfCNCPoint6[4672] = {X 137.4231, Y 19.8782, Z -8.0000, A 0.000, B 0.000, C 0.000 }
gfCNCPoint6[4673] = {X 136.8907, Y 20.5225, Z -8.0000, A 0.000, B 0.000, C 0.000 }
gfCNCPoint6[4674] = {X 136.2442, Y 21.0523, Z -8.0000, A 0.000, B 0.000, C 0.000 }
gfCNCPoint6[4675] = {X 135.5078, Y 21.4476, Z -8.0000, A 0.000, B 0.000, C 0.000 }
gfCNCPoint6[4676] = {X 134.7090, Y 21.6937, Z -8.0000, A 0.000, B 0.000, C 0.000 }
gfCNCPoint6[4677] = {X 133.8778, Y 21.7814, Z -8.0000, A 0.000, B 0.000, C 0.000 }
gfCNCPoint6[4678] = {X 133.2006, Y 21.7815, Z -8.0000, A 0.000, B 0.000, C 0.000 }
gfCNCPoint6[4679] = {X 132.2394, Y 21.6732, Z -8.0000, A 0.000, B 0.000, C 0.000 }
gfCNCPoint6[4680] = {X 131.3263, Y 21.3537, Z -8.0000, A 0.000, B 0.000, C 0.000 }
gfCNCPoint6[4681] = {X 130.5072, Y 20.8390, Z -8.0000, A 0.000, B 0.000, C 0.000 }
gfCNCPoint6[4682] = {X 129.8231, Y 20.1550, Z -8.0000, A 0.000, B 0.000, C 0.000 }
gfCNCPoint6[4683] = {X 129.3085, Y 19.3359, Z -8.0000, A 0.000, B 0.000, C 0.000 }
gfCNCPoint6[4684] = {X 128.9890, Y 18.4228, Z -8.0000, A 0.000, B 0.000, C 0.000 }
gfCNCPoint6[4685] = {X 128.8806, Y 17.4615, Z -8.0000, A 0.000, B 0.000, C 0.000 }
gfCNCPoint6[4686] = {X 128.8806, Y 10.4835, Z -8.0000, A 0.000, B 0.000, C 0.000 }
gfCNCPoint6[4687] = {X 128.9874, Y 9.5289, Z -8.0000, A 0.000, B 0.000, C 0.000 }
gfCNCPoint6[4688] = {X 129.3026, Y 8.6214, Z -8.0000, A 0.000, B 0.000, C 0.000 }
gfCNCPoint6[4689] = {X 129.8104, Y 7.8061, Z -8.0000, A 0.000, B 0.000, C 0.000 }
gfCNCPoint6[4690] = {X 130.4859, Y 7.1231, Z -8.0000, A 0.000, B 0.000, C 0.000 }
gfCNCPoint6[4691] = {X 131.2956, Y 6.6063, Z -8.0000, A 0.000, B 0.000, C 0.000 }
gfCNCPoint6[4692] = {X 132.1995, Y 6.2811, Z -8.0000, A 0.000, B 0.000, C 0.000 }
gfCNCPoint6[4693] = {X 133.1529, Y 6.1638, Z -8.0000, A 0.000, B 0.000, C 0.000 }
gfCNCPoint6[4694] = {X 133.8866, Y 6.1637, Z -8.0000, A 0.000, B 0.000, C 0.000 }
gfCNCPoint6[4695] = {X 134.7107, Y 6.2517, Z -8.0000, A 0.000, B 0.000, C 0.000 }
gfCNCPoint6[4696] = {X 135.5029, Y 6.4954, Z -8.0000, A 0.000, B 0.000, C 0.000 }
gfCNCPoint6[4697] = {X 136.2340, Y 6.8860, Z -8.0000, A 0.000, B 0.000, C 0.000 }
gfCNCPoint6[4698] = {X 136.8770, Y 7.4089, Z -8.0000, A 0.000, B 0.000, C 0.000 }
gfCNCPoint6[4699] = {X 137.4083, Y 8.0450, Z -8.0000, A 0.000, B 0.000, C 0.000 }
gfCNCPoint6[4700] = {X 155.1135, Y 8.0464, Z -8.0000, A 0.000, B 0.000, C 0.000 }
gfCNCPoint6[4701] = {X 155.6455, Y 7.4091, Z -8.0000, A 0.000, B 0.000, C 0.000 }
gfCNCPoint6[4702] = {X 156.2896, Y 6.8854, Z -8.0000, A 0.000, B 0.000, C 0.000 }
gfCNCPoint6[4703] = {X 157.0220, Y 6.4945, Z -8.0000, A 0.000, B 0.000, C 0.000 }
gfCNCPoint6[4704] = {X 157.8157, Y 6.2510, Z -8.0000, A 0.000, B 0.000, C 0.000 }
gfCNCPoint6[4705] = {X 158.6412, Y 6.1637, Z -8.0000, A 0.000, B 0.000, C 0.000 }
gfCNCPoint6[4706] = {X 159.3781, Y 6.1639, Z -8.0000, A 0.000, B 0.000, C 0.000 }
gfCNCPoint6[4707] = {X 160.3301, Y 6.2828, Z -8.0000, A 0.000, B 0.000, C 0.000 }
gfCNCPoint6[4708] = {X 161.2324, Y 6.6088, Z -8.0000, A 0.000, B 0.000, C 0.000 }
gfCNCPoint6[4709] = {X 162.0405, Y 7.1260, Z -8.0000, A 0.000, B 0.000, C 0.000 }
gfCNCPoint6[4710] = {X 162.7145, Y 7.8088, Z -8.0000, A 0.000, B 0.000, C 0.000 }
gfCNCPoint6[4711] = {X 163.2212, Y 8.6236, Z -8.0000, A 0.000, B 0.000, C 0.000 }
gfCNCPoint6[4712] = {X 163.5355, Y 9.5300, Z -8.0000, A 0.000, B 0.000, C 0.000 }
gfCNCPoint6[4713] = {X 163.6421, Y 10.4835, Z -8.0000, A 0.000, B 0.000, C 0.000 }
gfCNCPoint6[4714] = {X 163.6421, Y 17.4615, Z -8.0000, A 0.000, B 0.000, C 0.000 }
gfCNCPoint6[4715] = {X 163.5355, Y 18.4152, Z -8.0000, A 0.000, B 0.000, C 0.000 }
gfCNCPoint6[4716] = {X 163.2211, Y 19.3218, Z -8.0000, A 0.000, B 0.000, C 0.000 }
gfCNCPoint6[4717] = {X 162.7142, Y 20.1366, Z -8.0000, A 0.000, B 0.000, C 0.000 }
gfCNCPoint6[4718] = {X 162.0400, Y 20.8194, Z -8.0000, A 0.000, B 0.000, C 0.000 }
gfCNCPoint6[4719] = {X 161.2318, Y 21.3365, Z -8.0000, A 0.000, B 0.000, C 0.000 }
gfCNCPoint6[4720] = {X 160.3292, Y 21.6625, Z -8.0000, A 0.000, B 0.000, C 0.000 }
gfCNCPoint6[4721] = {X 159.3770, Y 21.7812, Z -8.0000, A 0.000, B 0.000, C 0.000 }
gfCNCPoint6[4722] = {X 158.6795, Y 21.7815, Z -8.0000, A 0.000, B 0.000, C 0.000 }
gfCNCPoint6[4723] = {X 157.8410, Y 21.6972, Z -8.0000, A 0.000, B 0.000, C 0.000 }
gfCNCPoint6[4724] = {X 157.0346, Y 21.4528, Z -8.0000, A 0.000, B 0.000, C 0.000 }
gfCNCPoint6[4725] = {X 156.2904, Y 21.0574, Z -8.0000, A 0.000, B 0.000, C 0.000 }
gfCNCPoint6[4726] = {X 155.6365, Y 20.5259, Z -8.0000, A 0.000, B 0.000, C 0.000 }
gfCNCPoint6[4727] = {X 155.0973, Y 19.8783, Z -8.0000, A 0.000, B 0.000, C 0.000 }
gfCNCPoint6[4728] = {X 152.2774, Y 19.8791, Z -8.0000, A 0.000, B 0.000, C 0.000 }
gfCNCPoint6[4729] = {X 152.2764, Y 40.8742, Z -8.0000, A 0.000, B 0.000, C 0.000 }
gfCNCPoint6[4730] = {X 152.7408, Y 41.3742, Z -8.0000, A 0.000, B 0.000, C 0.000 }
gfCNCPoint6[4731] = {X 152.8370, Y 41.4886, Z -8.0000, A 0.000, B 0.000, C 0.000 }
gfCNCPoint6[4732] = {X 153.3627, Y 42.3139, Z -8.0000, A 0.000, B 0.000, C 0.000 }
gfCNCPoint6[4733] = {X 153.6903, Y 43.2360, Z -8.0000, A 0.000, B 0.000, C 0.000 }
gfCNCPoint6[4734] = {X 153.8031, Y 44.2080, Z -8.0000, A 0.000, B 0.000, C 0.000 }
gfCNCPoint6[4735] = {X 153.8029, Y 45.0415, Z -8.0000, A 0.000, B 0.000, C 0.000 }
gfCNCPoint6[4736] = {X 153.6867, Y 45.9960, Z -8.0000, A 0.000, B 0.000, C 0.000 }
gfCNCPoint6[4737] = {X 153.3623, Y 46.9011, Z -8.0000, A 0.000, B 0.000, C 0.000 }
gfCNCPoint6[4738] = {X 152.8458, Y 47.7120, Z -8.0000, A 0.000, B 0.000, C 0.000 }
gfCNCPoint6[4739] = {X 152.1626, Y 48.3886, Z -8.0000, A 0.000, B 0.000, C 0.000 }
gfCNCPoint6[4740] = {X 151.3468, Y 48.8973, Z -8.0000, A 0.000, B 0.000, C 0.000 }
gfCNCPoint6[4741] = {X 150.4386, Y 49.2130, Z -8.0000, A 0.000, B 0.000, C 0.000 }
gfCNCPoint6[4742] = {X 149.4831, Y 49.3200, Z -8.0000, A 0.000, B 0.000, C 0.000 }
gfCNCPoint6[4743] = {X 143.0396, Y 49.3200, Z -8.0000, A 0.000, B 0.000, C 0.000 }
gfCNCPoint6[4744] = {X 142.0831, Y 49.2128, Z -8.0000, A 0.000, B 0.000, C 0.000 }
gfCNCPoint6[4745] = {X 141.1741, Y 48.8964, Z -8.0000, A 0.000, B 0.000, C 0.000 }
gfCNCPoint6[4746] = {X 140.3576, Y 48.3866, Z -8.0000, A 0.000, B 0.000, C 0.000 }
gfCNCPoint6[4747] = {X 139.6743, Y 47.7087, Z -8.0000, A 0.000, B 0.000, C 0.000 }
gfCNCPoint6[4748] = {X 139.1581, Y 46.8964, Z -8.0000, A 0.000, B 0.000, C 0.000 }
gfCNCPoint6[4749] = {X 138.8346, Y 45.9899, Z -8.0000, A 0.000, B 0.000, C 0.000 }
gfCNCPoint6[4750] = {X 138.7198, Y 45.0342, Z -8.0000, A 0.000, B 0.000, C 0.000 }
gfCNCPoint6[4751] = {X 138.7200, Y 44.1494, Z -8.0000, A 0.000, B 0.000, C 0.000 }
gfCNCPoint6[4752] = {X 138.8305, Y 43.2364, Z -8.0000, A 0.000, B 0.000, C 0.000 }
gfCNCPoint6[4753] = {X 139.1317, Y 42.3675, Z -8.0000, A 0.000, B 0.000, C 0.000 }
gfCNCPoint6[4754] = {X 139.6099, Y 41.5821, Z -8.0000, A 0.000, B 0.000, C 0.000 }
gfCNCPoint6[4755] = {X 140.2436, Y 40.9157, Z -8.0000, A 0.000, B 0.000, C 0.000 }
gfCNCPoint6[4756] = {X 140.2436, Y 30.3971, Z -8.0000, A 0.000, B 0.000, C 0.000 }
gfCNCPoint6[4757] = {X 136.2436, Y 30.3971, Z -8.0000, A 0.000, B 0.000, C 0.000 }
gfCNCPoint6[4758] = {X 140.3236, Y 30.3971, Z -8.0000, A 0.000, B 0.000, C 0.000 }
gfCNCPoint6[4759] = {X 140.3236, Y 19.7985, Z -8.0000, A 0.000, B 0.000, C 0.000 }
gfCNCPoint6[4760] = {X 137.3791, Y 19.7982, Z -8.0000, A 0.000, B 0.000, C 0.000 }
gfCNCPoint6[4761] = {X 137.3563, Y 19.8342, Z -8.0000, A 0.000, B 0.000, C 0.000 }
gfCNCPoint6[4762] = {X 136.8338, Y 20.4663, Z -8.0000, A 0.000, B 0.000, C 0.000 }
gfCNCPoint6[4763] = {X 136.1993, Y 20.9861, Z -8.0000, A 0.000, B 0.000, C 0.000 }
gfCNCPoint6[4764] = {X 135.4766, Y 21.3739, Z -8.0000, A 0.000, B 0.000, C 0.000 }
gfCNCPoint6[4765] = {X 134.6928, Y 21.6154, Z -8.0000, A 0.000, B 0.000, C 0.000 }
gfCNCPoint6[4766] = {X 133.8772, Y 21.7014, Z -8.0000, A 0.000, B 0.000, C 0.000 }
gfCNCPoint6[4767] = {X 133.2006, Y 21.7015, Z -8.0000, A 0.000, B 0.000, C 0.000 }
gfCNCPoint6[4768] = {X 132.2572, Y 21.5952, Z -8.0000, A 0.000, B 0.000, C 0.000 }
gfCNCPoint6[4769] = {X 131.3610, Y 21.2816, Z -8.0000, A 0.000, B 0.000, C 0.000 }
gfCNCPoint6[4770] = {X 130.5570, Y 20.7765, Z -8.0000, A 0.000, B 0.000, C 0.000 }
gfCNCPoint6[4771] = {X 129.8857, Y 20.1051, Z -8.0000, A 0.000, B 0.000, C 0.000 }
gfCNCPoint6[4772] = {X 129.3805, Y 19.3012, Z -8.0000, A 0.000, B 0.000, C 0.000 }
gfCNCPoint6[4773] = {X 129.0669, Y 18.4050, Z -8.0000, A 0.000, B 0.000, C 0.000 }
gfCNCPoint6[4774] = {X 128.9606, Y 17.4615, Z -8.0000, A 0.000, B 0.000, C 0.000 }
gfCNCPoint6[4775] = {X 128.9606, Y 10.4835, Z -8.0000, A 0.000, B 0.000, C 0.000 }
gfCNCPoint6[4776] = {X 129.0655, Y 9.5466, Z -8.0000, A 0.000, B 0.000, C 0.000 }
gfCNCPoint6[4777] = {X 129.3747, Y 8.6559, Z -8.0000, A 0.000, B 0.000, C 0.000 }
gfCNCPoint6[4778] = {X 129.8732, Y 7.8557, Z -8.0000, A 0.000, B 0.000, C 0.000 }
gfCNCPoint6[4779] = {X 130.5362, Y 7.1853, Z -8.0000, A 0.000, B 0.000, C 0.000 }
gfCNCPoint6[4780] = {X 131.3309, Y 6.6781, Z -8.0000, A 0.000, B 0.000, C 0.000 }
gfCNCPoint6[4781] = {X 132.2180, Y 6.3589, Z -8.0000, A 0.000, B 0.000, C 0.000 }
gfCNCPoint6[4782] = {X 133.1538, Y 6.2438, Z -8.0000, A 0.000, B 0.000, C 0.000 }
gfCNCPoint6[4783] = {X 133.8858, Y 6.2437, Z -8.0000, A 0.000, B 0.000, C 0.000 }
gfCNCPoint6[4784] = {X 134.7029, Y 6.3318, Z -8.0000, A 0.000, B 0.000, C 0.000 }
gfCNCPoint6[4785] = {X 135.4877, Y 6.5758, Z -8.0000, A 0.000, B 0.000, C 0.000 }
gfCNCPoint6[4786] = {X 136.2106, Y 6.9666, Z -8.0000, A 0.000, B 0.000, C 0.000 }
gfCNCPoint6[4787] = {X 136.8446, Y 7.4896, Z -8.0000, A 0.000, B 0.000, C 0.000 }
gfCNCPoint6[4788] = {X 137.3658, Y 8.1250, Z -8.0000, A 0.000, B 0.000, C 0.000 }
gfCNCPoint6[4789] = {X 155.1560, Y 8.1264, Z -8.0000, A 0.000, B 0.000, C 0.000 }
gfCNCPoint6[4790] = {X 155.6779, Y 7.4898, Z -8.0000, A 0.000, B 0.000, C 0.000 }
gfCNCPoint6[4791] = {X 156.3129, Y 6.9661, Z -8.0000, A 0.000, B 0.000, C 0.000 }
gfCNCPoint6[4792] = {X 157.0372, Y 6.5749, Z -8.0000, A 0.000, B 0.000, C 0.000 }
gfCNCPoint6[4793] = {X 157.8234, Y 6.3310, Z -8.0000, A 0.000, B 0.000, C 0.000 }
gfCNCPoint6[4794] = {X 158.6420, Y 6.2437, Z -8.0000, A 0.000, B 0.000, C 0.000 }
gfCNCPoint6[4795] = {X 159.3770, Y 6.2439, Z -8.0000, A 0.000, B 0.000, C 0.000 }
gfCNCPoint6[4796] = {X 160.3114, Y 6.3606, Z -8.0000, A 0.000, B 0.000, C 0.000 }
gfCNCPoint6[4797] = {X 161.1970, Y 6.6806, Z -8.0000, A 0.000, B 0.000, C 0.000 }
gfCNCPoint6[4798] = {X 161.9902, Y 7.1882, Z -8.0000, A 0.000, B 0.000, C 0.000 }
gfCNCPoint6[4799] = {X 162.6517, Y 7.8584, Z -8.0000, A 0.000, B 0.000, C 0.000 }
gfCNCPoint6[4800] = {X 163.1490, Y 8.6580, Z -8.0000, A 0.000, B 0.000, C 0.000 }
gfCNCPoint6[4801] = {X 163.4575, Y 9.5477, Z -8.0000, A 0.000, B 0.000, C 0.000 }
gfCNCPoint6[4802] = {X 163.5621, Y 10.4835, Z -8.0000, A 0.000, B 0.000, C 0.000 }
gfCNCPoint6[4803] = {X 163.5621, Y 17.4615, Z -8.0000, A 0.000, B 0.000, C 0.000 }
gfCNCPoint6[4804] = {X 163.4575, Y 18.3975, Z -8.0000, A 0.000, B 0.000, C 0.000 }
gfCNCPoint6[4805] = {X 163.1489, Y 19.2873, Z -8.0000, A 0.000, B 0.000, C 0.000 }
gfCNCPoint6[4806] = {X 162.6514, Y 20.0870, Z -8.0000, A 0.000, B 0.000, C 0.000 }
gfCNCPoint6[4807] = {X 161.9897, Y 20.7572, Z -8.0000, A 0.000, B 0.000, C 0.000 }
gfCNCPoint6[4808] = {X 161.1964, Y 21.2648, Z -8.0000, A 0.000, B 0.000, C 0.000 }
gfCNCPoint6[4809] = {X 160.3106, Y 21.5847, Z -8.0000, A 0.000, B 0.000, C 0.000 }
gfCNCPoint6[4810] = {X 159.3760, Y 21.7012, Z -8.0000, A 0.000, B 0.000, C 0.000 }
gfCNCPoint6[4811] = {X 158.6797, Y 21.7015, Z -8.0000, A 0.000, B 0.000, C 0.000 }
gfCNCPoint6[4812] = {X 157.8484, Y 21.6171, Z -8.0000, A 0.000, B 0.000, C 0.000 }
gfCNCPoint6[4813] = {X 157.0495, Y 21.3724, Z -8.0000, A 0.000, B 0.000, C 0.000 }
gfCNCPoint6[4814] = {X 156.3135, Y 20.9766, Z -8.0000, A 0.000, B 0.000, C 0.000 }
gfCNCPoint6[4815] = {X 155.6688, Y 20.4452, Z -8.0000, A 0.000, B 0.000, C 0.000 }
gfCNCPoint6[4816] = {X 155.1399, Y 19.7982, Z -8.0000, A 0.000, B 0.000, C 0.000 }
gfCNCPoint6[4817] = {X 152.1974, Y 19.7991, Z -8.0000, A 0.000, B 0.000, C 0.000 }
gfCNCPoint6[4818] = {X 152.1964, Y 40.9056, Z -8.0000, A 0.000, B 0.000, C 0.000 }
gfCNCPoint6[4819] = {X 152.6808, Y 41.4271, Z -8.0000, A 0.000, B 0.000, C 0.000 }
gfCNCPoint6[4820] = {X 152.7753, Y 41.5395, Z -8.0000, A 0.000, B 0.000, C 0.000 }
gfCNCPoint6[4821] = {X 153.2911, Y 42.3495, Z -8.0000, A 0.000, B 0.000, C 0.000 }
gfCNCPoint6[4822] = {X 153.6124, Y 43.2544, Z -8.0000, A 0.000, B 0.000, C 0.000 }
gfCNCPoint6[4823] = {X 153.7231, Y 44.2082, Z -8.0000, A 0.000, B 0.000, C 0.000 }
gfCNCPoint6[4824] = {X 153.7229, Y 45.0408, Z -8.0000, A 0.000, B 0.000, C 0.000 }
gfCNCPoint6[4825] = {X 153.6089, Y 45.9775, Z -8.0000, A 0.000, B 0.000, C 0.000 }
gfCNCPoint6[4826] = {X 153.2905, Y 46.8659, Z -8.0000, A 0.000, B 0.000, C 0.000 }
gfCNCPoint6[4827] = {X 152.7835, Y 47.6618, Z -8.0000, A 0.000, B 0.000, C 0.000 }
gfCNCPoint6[4828] = {X 152.1130, Y 48.3258, Z -8.0000, A 0.000, B 0.000, C 0.000 }
gfCNCPoint6[4829] = {X 151.3123, Y 48.8251, Z -8.0000, A 0.000, B 0.000, C 0.000 }
gfCNCPoint6[4830] = {X 150.4209, Y 49.1350, Z -8.0000, A 0.000, B 0.000, C 0.000 }
gfCNCPoint6[4831] = {X 149.4831, Y 49.2400, Z -8.0000, A 0.000, B 0.000, C 0.000 }
gfCNCPoint6[4832] = {X 143.0396, Y 49.2400, Z -8.0000, A 0.000, B 0.000, C 0.000 }
gfCNCPoint6[4833] = {X 142.1008, Y 49.1348, Z -8.0000, A 0.000, B 0.000, C 0.000 }
gfCNCPoint6[4834] = {X 141.2086, Y 48.8243, Z -8.0000, A 0.000, B 0.000, C 0.000 }
gfCNCPoint6[4835] = {X 140.4073, Y 48.3239, Z -8.0000, A 0.000, B 0.000, C 0.000 }
gfCNCPoint6[4836] = {X 139.7367, Y 47.6586, Z -8.0000, A 0.000, B 0.000, C 0.000 }
gfCNCPoint6[4837] = {X 139.2300, Y 46.8612, Z -8.0000, A 0.000, B 0.000, C 0.000 }
gfCNCPoint6[4838] = {X 138.9124, Y 45.9715, Z -8.0000, A 0.000, B 0.000, C 0.000 }
gfCNCPoint6[4839] = {X 138.7998, Y 45.0336, Z -8.0000, A 0.000, B 0.000, C 0.000 }
gfCNCPoint6[4840] = {X 138.8000, Y 44.1505, Z -8.0000, A 0.000, B 0.000, C 0.000 }
gfCNCPoint6[4841] = {X 138.9105, Y 43.2454, Z -8.0000, A 0.000, B 0.000, C 0.000 }
gfCNCPoint6[4842] = {X 139.2119, Y 42.3850, Z -8.0000, A 0.000, B 0.000, C 0.000 }
gfCNCPoint6[4843] = {X 139.6903, Y 41.6088, Z -8.0000, A 0.000, B 0.000, C 0.000 }
gfCNCPoint6[4844] = {X 140.3236, Y 40.9529, Z -8.0000, A 0.000, B 0.000, C 0.000 }
gfCNCPoint6[4845] = {X 140.3236, Y 30.3971, Z -8.0000, A 0.000, B 0.000, C 0.000 }
gfCNCPoint6[4846] = {X 136.3236, Y 30.3971, Z -8.0000, A 0.000, B 0.000, C 0.000 }
gfCNCPoint6[4847] = {X 140.4036, Y 30.3971, Z -8.0000, A 0.000, B 0.000, C 0.000 }
gfCNCPoint6[4848] = {X 140.4036, Y 19.7185, Z -8.0000, A 0.000, B 0.000, C 0.000 }
gfCNCPoint6[4849] = {X 137.3351, Y 19.7182, Z -8.0000, A 0.000, B 0.000, C 0.000 }
gfCNCPoint6[4850] = {X 137.2894, Y 19.7904, Z -8.0000, A 0.000, B 0.000, C 0.000 }
gfCNCPoint6[4851] = {X 136.7767, Y 20.4103, Z -8.0000, A 0.000, B 0.000, C 0.000 }
gfCNCPoint6[4852] = {X 136.1542, Y 20.9199, Z -8.0000, A 0.000, B 0.000, C 0.000 }
gfCNCPoint6[4853] = {X 135.4454, Y 21.3003, Z -8.0000, A 0.000, B 0.000, C 0.000 }
gfCNCPoint6[4854] = {X 134.6765, Y 21.5370, Z -8.0000, A 0.000, B 0.000, C 0.000 }
gfCNCPoint6[4855] = {X 133.8765, Y 21.6214, Z -8.0000, A 0.000, B 0.000, C 0.000 }
gfCNCPoint6[4856] = {X 133.2006, Y 21.6215, Z -8.0000, A 0.000, B 0.000, C 0.000 }
gfCNCPoint6[4857] = {X 132.2750, Y 21.5172, Z -8.0000, A 0.000, B 0.000, C 0.000 }
gfCNCPoint6[4858] = {X 131.3957, Y 21.2096, Z -8.0000, A 0.000, B 0.000, C 0.000 }
gfCNCPoint6[4859] = {X 130.6069, Y 20.7140, Z -8.0000, A 0.000, B 0.000, C 0.000 }
gfCNCPoint6[4860] = {X 129.9482, Y 20.0553, Z -8.0000, A 0.000, B 0.000, C 0.000 }
